REGION Network 4: Diagnostico ASi Global
   // solamente es esta llamada
   RUNG wire#powerrail
      I_Contact( "Activar_Simulador" )
      "FC953_Diagnostico_ASi"(Array_ASI3_C1 := "DB1903_ASI_DIAG".ASI3_GW_C1, Array_ASI3_C2 := "DB1903_ASI_DIAG".ASI3_GW_C2, Array_ASI5_Flags := "DB1903_ASI_DIAG".ASI5_GW_Flags, Error_ASI => "DB1903_ASI_DIAG".ASI_Gateway_Error)
   END_RUNG
   // the same network as SCL:
   IF NOT "Activar_Simulador" THEN
       "FC953_Diagnostico_ASi"(Array_ASI3_C1 := "DB1903_ASI_DIAG".ASI3_GW_C1,
                               Array_ASI3_C2 := "DB1903_ASI_DIAG".ASI3_GW_C2,
                               Array_ASI5_Flags := "DB1903_ASI_DIAG".ASI5_GW_Flags,
                               Error_ASI => "DB1903_ASI_DIAG".ASI_Gateway_Error);
   END_IF;
END_REGION
END_ORGANIZATION_BLOCK

ORGANIZATION_BLOCK "OB82_I/O_FLT1"   // OB82, LAD, DiagnosticErrorInterrupt
TITLE = "I/O Point Fault"
{ S7_Optimized_Access := 'FALSE' }
AUTHOR : ESTANDAR
VERSION : 3.0
// stored: SetENOAutomatically false
   VAR_TEMP
      OB82_EV_CLASS : Byte;   // 16#39, Event class 3, Entering event state, Internal fault event
      OB82_FLT_ID : Byte;   // 16#XX, Fault identifcation code
      OB82_PRIORITY : Byte;   // Priority of OB Execution
      OB82_OB_NUMBR : Byte;   // 82 (Organization block 82, OB82)
      OB82_RESERVED_1 : Byte;   // Reserved for system
      OB82_IO_FLAG : Byte;   // Input (01010100), Output (01010101)
      OB82_MDL_ADDR : Word;   // Base address of module with fault
      OB82_MDL_DEFECT : Bool;   // Module defective
      OB82_INT_FAULT : Bool;   // Internal fault
      OB82_EXT_FAULT : Bool;   // External fault
      OB82_PNT_INFO : Bool;   // Point information
      OB82_EXT_VOLTAGE : Bool;   // External voltage low
      OB82_FLD_CONNCTR : Bool;   // Field wiring connector missing
      OB82_NO_CONFIG : Bool;   // Module has no configuration data
      OB82_CONFIG_ERR : Bool;   // Module has configuration error
      OB82_MDL_TYPE : Byte;   // Type of module
      OB82_SUB_MDL_ERR : Bool;   // Sub-Module is missing or has error
      OB82_COMM_FAULT : Bool;   // Communication fault
      OB82_MDL_STOP : Bool;   // Module is stopped
      OB82_WTCH_DOG_FLT : Bool;   // Watch dog timer stopped module
      OB82_INT_PS_FLT : Bool;   // Internal power supply fault
      OB82_PRIM_BATT_FLT : Bool;   // Primary battery is in fault
      OB82_BCKUP_BATT_FLT : Bool;   // Backup battery is in fault
      OB82_RESERVED_2 : Bool;   // Reserved for system
      OB82_RACK_FLT : Bool;   // Rack fault, only for bus interface module
      OB82_PROC_FLT : Bool;   // Processor fault
      OB82_EPROM_FLT : Bool;   // EPROM fault
      OB82_RAM_FLT : Bool;   // RAM fault
      OB82_ADU_FLT : Bool;   // ADU fault
      OB82_FUSE_FLT : Bool;   // Fuse fault
      OB82_HW_INTR_FLT : Bool;   // Hardware interupt input in fault
      OB82_RESERVED_3 : Bool;   // Reserved for system
      OB82_DATE_TIME : Date_And_Time;   // Date and time OB82 started
   END_VAR
BEGIN
END_ORGANIZATION_BLOCK

ORGANIZATION_BLOCK "OB83_I/O_FLT2"   // OB83, LAD, PullOrPlugOfModules
TITLE = "I/O Point Fault"
{ S7_Optimized_Access := 'FALSE' }
// stored: SetENOAutomatically false
   VAR_TEMP
      OB83_EV_CLASS : Byte;   // 16#38/39, Event class 3, module inserted/removed (8/9)
      OB83_FLT_ID : Byte;   // 16#XX, Fault identifcation code
      OB83_PRIORITY : Byte;   // 26/28 (Priority of 1 is lowest)
      OB83_OB_NUMBR : Byte;   // 83 (Organization block 83, OB83)
      OB83_RESERVED_1 : Byte;   // Reserved for system
      OB83_MDL_ID : Byte;   // Input module (01010100), Output module (01010101)
      OB83_MDL_ADDR : Word;   // Base address of module with point fault
      OB83_RACK_NUM : Word;   // Number of rack that has module with point fault
      OB83_MDL_TYPE : Word;   // Module type with point fault
      OB83_DATE_TIME : Date_And_Time;   // Date and time OB83 started
   END_VAR
BEGIN
END_ORGANIZATION_BLOCK

ORGANIZATION_BLOCK "OB86_ERROR_SLAVES"   // OB86, LAD, RackOrStationFailure
TITLE = "Loss Of Rack Fault"
{ S7_Optimized_Access := 'FALSE' }
AUTHOR : ESTANDAR
VERSION : 3.0
// stored: SetENOAutomatically false
   VAR_TEMP
      OB86_EV_CLASS : Byte;   // 16#38/39 Event class 3
      OB86_FLT_ID : Byte;   // 16#C1/C4/C5, Fault identifcation code
      OB86_PRIORITY : Byte;   // Priority of OB Execution
      OB86_OB_NUMBR : Byte;   // 86 (Organization block 86, OB86)
      OB86_RESERVED_1 : Byte;   // Reserved for system
      OB86_RESERVED_2 : Byte;   // Reserved for system
      OB86_MDL_ADDR : Word;   // Base address of IM module in rack with fault
      OB86_Z23 : DWord;
      OB86_DATE_TIME : Date_And_Time;   // Date and time OB86 started
      P_destino : DWord;
      P_origen : DWord;
      P_infonodo : DWord;
      Numnodo : Word;
      Numred : Word;
      infonodo : Struct
         had_failed : Bool;
         deactivated : Bool;
         reserved_10 : Bool;
         reserved_11 : Bool;
         reserved_12 : Bool;
         reserved_13 : Bool;
         reserved_14 : Bool;
         reserved_15 : Bool;
         OK : Bool;
         maintenance : Bool;
         faulty : Bool;
         failed : Bool;
         was_deactivated : Bool;
         DPV1 : Bool;
         was_under_maintenance : Bool;
         was_failed : Bool;
      END_STRUCT;
   END_VAR
BEGIN
END_ORGANIZATION_BLOCK

FUNCTION_BLOCK "FB420_MesaTL_EtiquetaOrden"   // FB420, LAD
{ S7_Optimized_Access := 'FALSE' }
AUTHOR : ROUTER
NAME : 20180615
VERSION : 3.1
// stored: AutoNumber false, SetENOAutomatically false
   VAR_INPUT
      NumeroMesa : UInt;
      pHsMx : Bool;
      NumSCR : UInt;   // Numero de Scanner asociada a la mesa
      DBFIFO_SCR : UInt;   // DB de Etiquetas Leidas
      LongFIFO_SCR : UInt;   // Numero de Lecturas que se pueden Almacenar
      V_TmpEntrada : Time := T#500MS;
      V_TmpSalida : Time := T#1S;
      MesaDeJDT02 : Bool;
   END_VAR
   VAR_OUTPUT
      PermisoEntrada : Bool;
      PermisoSalida : Bool;
   END_VAR
   VAR
      Mx_ET00 : Bool;
      Mx_ET01 : Bool;
      Mx_ET02 : Bool;
      Mx_ET07 : Bool;
      Mx_ET10 : Bool;
      Mx_ET11 : Bool;
      Mx_ET12 : Bool;
      Mx_ET50 : Bool;
      Mx_ET51 : Bool;
      Mx_ET52 : Bool;
      PresenciaEmiOK : Bool;
      AusenciaEmiOK : Bool;
      BorradoOK : Bool;
      OrdenMx : UInt;
      Motivo : UInt;
      TmpEntrada { S7_SetPoint := 'True'} : TON_TIME;
      TmpSalida { S7_SetPoint := 'True'} : TON_TIME;
      Datos_Scanner { S7_SetPoint := 'True'} : "ROUT_Orden_Fifo_Scanner";
   END_VAR
   VAR_TEMP
      Aux_ET00 : Bool;
      ExisteOrdenSCR : Bool;
      SinOrdenSCR : Bool;
      ExisteOrdenMx : Bool;
      SinOrdenMx : Bool;
      Presencia : Bool;
      Ausencia : Bool;
      Ausencia_especial : Bool;
      MirarOrden : Bool;
      BorradoOrden : Bool;
      Emi_presencia : Bool;
      Emi_ausencia : Bool;
      MesaTMP : UInt;
      MotivoTMP : UInt;
      posicion : Int;
      i : Int;
      longitud : Int;
      codigo_string : String[20];
      mesa_string : String[5];
      moti_string : String[4];
      Mensaje_completo : String;
   END_VAR
BEGIN

REGION Network 1: Incializaciones de la Función
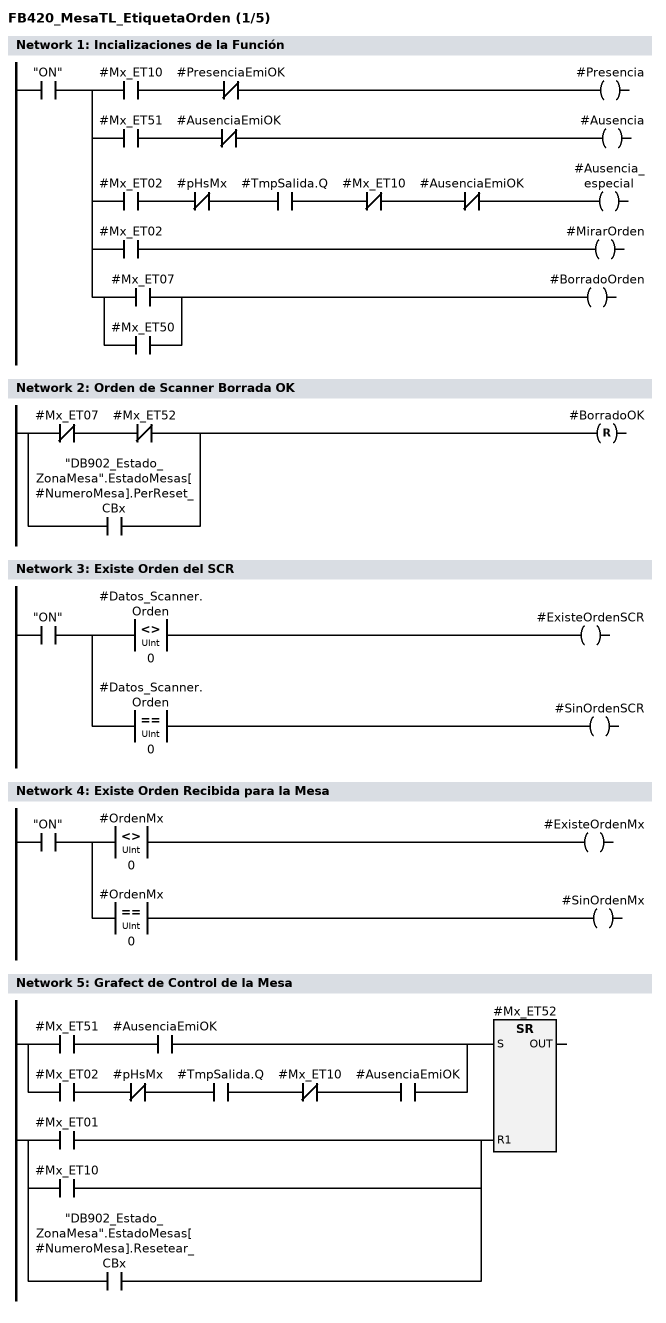
   RUNG wire#powerrail
      Contact( "ON" )
      wire#w1
      Contact( #Mx_ET10 )
      I_Contact( #PresenciaEmiOK )
      Coil( #Presencia )
   END_RUNG
   RUNG wire#w1
      Contact( #Mx_ET51 )
      I_Contact( #AusenciaEmiOK )
      Coil( #Ausencia )
   END_RUNG
   RUNG wire#w1
      Contact( #Mx_ET02 )
      I_Contact( #pHsMx )
      Contact( #TmpSalida.Q )
      I_Contact( #Mx_ET10 )
      I_Contact( #AusenciaEmiOK )
      Coil( #Ausencia_especial )
   END_RUNG
   RUNG wire#w1
      Contact( #Mx_ET02 )
      Coil( #MirarOrden )
   END_RUNG
   RUNG wire#w1
      Contact( #Mx_ET07 )
      wire#w2
      Coil( #BorradoOrden )
   END_RUNG
   RUNG wire#w1
      Contact( #Mx_ET50 )
   END_RUNG wire#w2
   // the same network as SCL:
   #Presencia := "ON" AND #Mx_ET10 AND NOT #PresenciaEmiOK;
   #Ausencia := "ON" AND #Mx_ET51 AND NOT #AusenciaEmiOK;
   #Ausencia_especial := "ON" AND #Mx_ET02 AND NOT #pHsMx AND #TmpSalida.Q AND NOT #Mx_ET10 AND NOT #AusenciaEmiOK;
   #MirarOrden := "ON" AND #Mx_ET02;
   #BorradoOrden := "ON" AND (#Mx_ET07 OR #Mx_ET50);
END_REGION

REGION Network 2: Orden de Scanner Borrada OK
   RUNG wire#powerrail
      I_Contact( #Mx_ET07 )
      I_Contact( #Mx_ET52 )
      wire#w1
      R_Coil( #BorradoOK )
   END_RUNG
   RUNG wire#powerrail
      Contact( "DB902_Estado_ZonaMesa".EstadoMesas[#NumeroMesa].PerReset_CBx )
   END_RUNG wire#w1
   // the same network as SCL:
   IF (NOT #Mx_ET07 AND NOT #Mx_ET52) OR "DB902_Estado_ZonaMesa".EstadoMesas[#NumeroMesa].PerReset_CBx THEN
       #BorradoOK := FALSE;
   END_IF;
END_REGION

REGION Network 3: Existe Orden del SCR
   RUNG wire#powerrail
      Contact( "ON" )
      wire#w1
      { S7_Templates := "SrcType := UInt" } NE_Contact(in1 := #Datos_Scanner.Orden, in2 := 0)
      Coil( #ExisteOrdenSCR )
   END_RUNG
   RUNG wire#w1
      { S7_Templates := "SrcType := UInt" } EQ_Contact(in1 := #Datos_Scanner.Orden, in2 := 0)
      Coil( #SinOrdenSCR )
   END_RUNG
   // the same network as SCL:
   #ExisteOrdenSCR := "ON" AND (#Datos_Scanner.Orden <> 0);
   #SinOrdenSCR := "ON" AND (#Datos_Scanner.Orden = 0);
END_REGION

REGION Network 4: Existe Orden Recibida para la Mesa
   RUNG wire#powerrail
      Contact( "ON" )
      wire#w1
      { S7_Templates := "SrcType := UInt" } NE_Contact(in1 := #OrdenMx, in2 := 0)
      Coil( #ExisteOrdenMx )
   END_RUNG
   RUNG wire#w1
      { S7_Templates := "SrcType := UInt" } EQ_Contact(in1 := #OrdenMx, in2 := 0)
      Coil( #SinOrdenMx )
   END_RUNG
   // the same network as SCL:
   #ExisteOrdenMx := "ON" AND (#OrdenMx <> 0);
   #SinOrdenMx := "ON" AND (#OrdenMx = 0);
END_REGION

REGION Network 5: Grafect de Control de la Mesa
   RUNG wire#powerrail
      Contact( #Mx_ET51 )
      Contact( #AusenciaEmiOK )
      wire#w1
      S_SR(operand := #Mx_ET52, r1 := wire#w2)
   END_RUNG
   RUNG wire#powerrail
      Contact( #Mx_ET02 )
      I_Contact( #pHsMx )
      Contact( #TmpSalida.Q )
      I_Contact( #Mx_ET10 )
      Contact( #AusenciaEmiOK )
   END_RUNG wire#w1
   RUNG wire#powerrail
      Contact( #Mx_ET01 )
   END_RUNG wire#w2
   RUNG wire#powerrail
      Contact( #Mx_ET10 )
   END_RUNG wire#w2
   RUNG wire#powerrail
      Contact( "DB902_Estado_ZonaMesa".EstadoMesas[#NumeroMesa].Resetear_CBx )
   END_RUNG wire#w2
   // the same network as SCL:
   IF (#Mx_ET51 AND #AusenciaEmiOK) OR (#Mx_ET02 AND NOT #pHsMx AND #TmpSalida.Q AND NOT #Mx_ET10 AND #AusenciaEmiOK) THEN
       #Mx_ET52 := TRUE;   // SR flip-flop
   END_IF;
   IF #Mx_ET01 OR #Mx_ET10 OR "DB902_Estado_ZonaMesa".EstadoMesas[#NumeroMesa].Resetear_CBx THEN
       #Mx_ET52 := FALSE;
   END_IF;
END_REGION

REGION Network 6
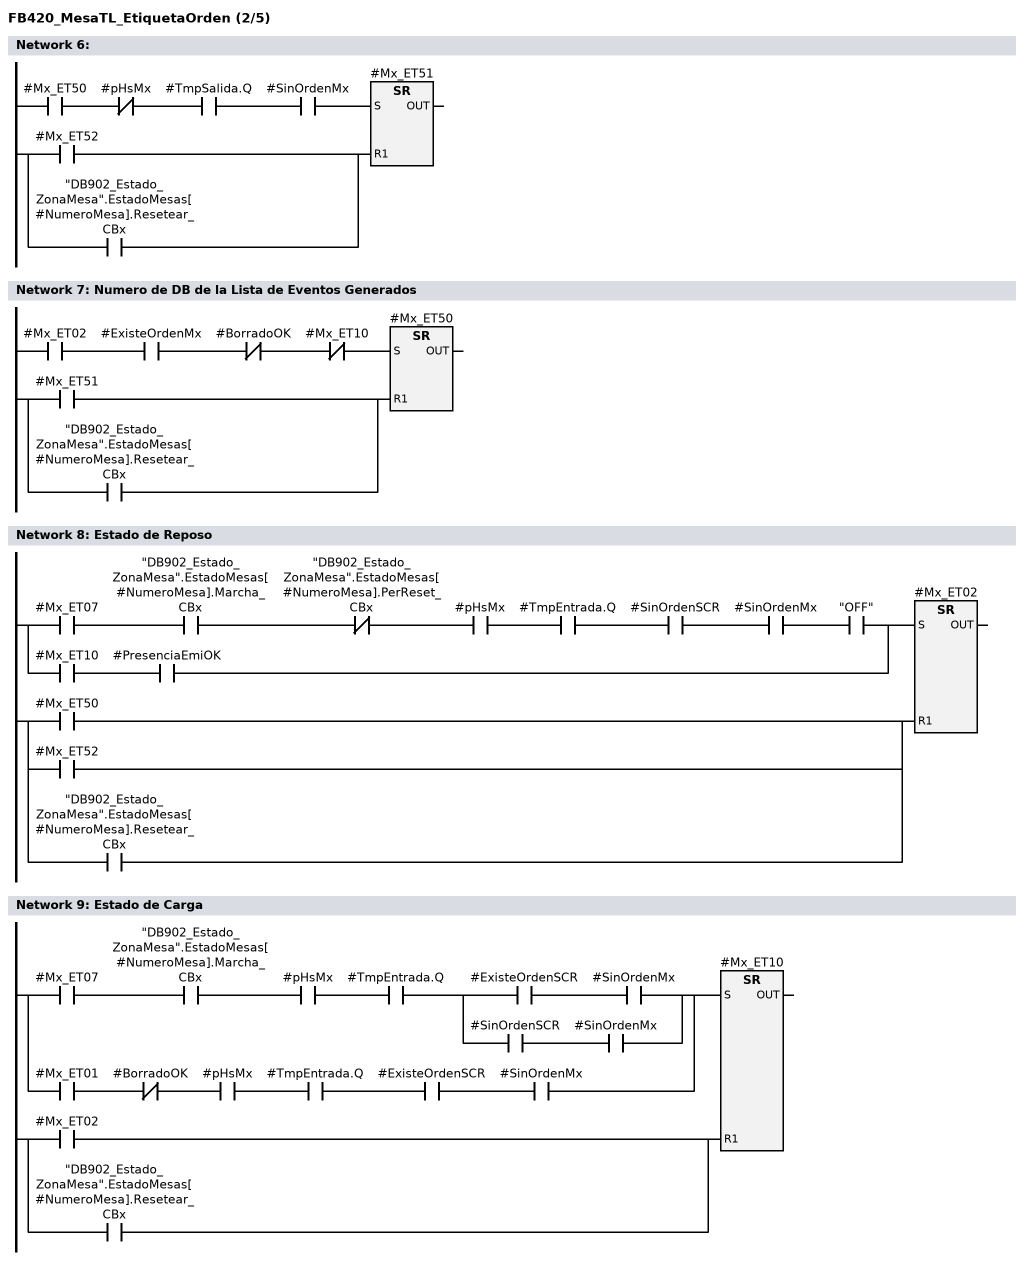
   RUNG wire#powerrail
      Contact( #Mx_ET50 )
      I_Contact( #pHsMx )
      Contact( #TmpSalida.Q )
      Contact( #SinOrdenMx )
      S_SR(operand := #Mx_ET51, r1 := wire#w1)
   END_RUNG
   RUNG wire#powerrail
      Contact( #Mx_ET52 )
   END_RUNG wire#w1
   RUNG wire#powerrail
      Contact( "DB902_Estado_ZonaMesa".EstadoMesas[#NumeroMesa].Resetear_CBx )
   END_RUNG wire#w1
   // the same network as SCL:
   IF #Mx_ET50 AND NOT #pHsMx AND #TmpSalida.Q AND #SinOrdenMx THEN
       #Mx_ET51 := TRUE;   // SR flip-flop
   END_IF;
   IF #Mx_ET52 OR "DB902_Estado_ZonaMesa".EstadoMesas[#NumeroMesa].Resetear_CBx THEN
       #Mx_ET51 := FALSE;
   END_IF;
END_REGION

REGION Network 7: Numero de DB de la Lista de Eventos Generados
   RUNG wire#powerrail
      Contact( #Mx_ET02 )
      Contact( #ExisteOrdenMx )
      I_Contact( #BorradoOK )
      I_Contact( #Mx_ET10 )
      S_SR(operand := #Mx_ET50, r1 := wire#w1)
   END_RUNG
   RUNG wire#powerrail
      Contact( #Mx_ET51 )
   END_RUNG wire#w1
   RUNG wire#powerrail
      Contact( "DB902_Estado_ZonaMesa".EstadoMesas[#NumeroMesa].Resetear_CBx )
   END_RUNG wire#w1
   // the same network as SCL:
   IF #Mx_ET02 AND #ExisteOrdenMx AND NOT #BorradoOK AND NOT #Mx_ET10 THEN
       #Mx_ET50 := TRUE;   // SR flip-flop
   END_IF;
   IF #Mx_ET51 OR "DB902_Estado_ZonaMesa".EstadoMesas[#NumeroMesa].Resetear_CBx THEN
       #Mx_ET50 := FALSE;
   END_IF;
END_REGION

REGION Network 8: Estado de Reposo
   RUNG wire#powerrail
      Contact( #Mx_ET07 )
      Contact( "DB902_Estado_ZonaMesa".EstadoMesas[#NumeroMesa].Marcha_CBx )
      I_Contact( "DB902_Estado_ZonaMesa".EstadoMesas[#NumeroMesa].PerReset_CBx )
      Contact( #pHsMx )
      Contact( #TmpEntrada.Q )
      Contact( #SinOrdenSCR )
      Contact( #SinOrdenMx )
      Contact( "OFF" )
      wire#w1
      S_SR(operand := #Mx_ET02, r1 := wire#w2)
   END_RUNG
   RUNG wire#powerrail
      Contact( #Mx_ET10 )
      Contact( #PresenciaEmiOK )
   END_RUNG wire#w1
   RUNG wire#powerrail
      Contact( #Mx_ET50 )
   END_RUNG wire#w2
   RUNG wire#powerrail
      Contact( #Mx_ET52 )
   END_RUNG wire#w2
   RUNG wire#powerrail
      Contact( "DB902_Estado_ZonaMesa".EstadoMesas[#NumeroMesa].Resetear_CBx )
   END_RUNG wire#w2
   // the same network as SCL:
   IF (#Mx_ET07 AND "DB902_Estado_ZonaMesa".EstadoMesas[#NumeroMesa].Marcha_CBx AND NOT "DB902_Estado_ZonaMesa".EstadoMesas[#NumeroMesa].PerReset_CBx AND #pHsMx AND #TmpEntrada.Q AND #SinOrdenSCR AND #SinOrdenMx AND "OFF") OR (#Mx_ET10 AND #PresenciaEmiOK) THEN
       #Mx_ET02 := TRUE;   // SR flip-flop
   END_IF;
   IF #Mx_ET50 OR #Mx_ET52 OR "DB902_Estado_ZonaMesa".EstadoMesas[#NumeroMesa].Resetear_CBx THEN
       #Mx_ET02 := FALSE;
   END_IF;
END_REGION

REGION Network 9: Estado de Carga
   RUNG wire#powerrail
      Contact( #Mx_ET07 )
      Contact( "DB902_Estado_ZonaMesa".EstadoMesas[#NumeroMesa].Marcha_CBx )
      Contact( #pHsMx )
      Contact( #TmpEntrada.Q )
      wire#w1
      Contact( #ExisteOrdenSCR )
      Contact( #SinOrdenMx )
      wire#w2
      S_SR(operand := #Mx_ET10, r1 := wire#w3)
   END_RUNG
   RUNG wire#w1
      Contact( #SinOrdenSCR )
      Contact( #SinOrdenMx )
   END_RUNG wire#w2
   RUNG wire#powerrail
      Contact( #Mx_ET01 )
      I_Contact( #BorradoOK )
      Contact( #pHsMx )
      Contact( #TmpEntrada.Q )
      Contact( #ExisteOrdenSCR )
      Contact( #SinOrdenMx )
   END_RUNG wire#w2
   RUNG wire#powerrail
      Contact( #Mx_ET02 )
   END_RUNG wire#w3
   RUNG wire#powerrail
      Contact( "DB902_Estado_ZonaMesa".EstadoMesas[#NumeroMesa].Resetear_CBx )
   END_RUNG wire#w3
   // the same network as SCL:
   IF (#Mx_ET07 AND "DB902_Estado_ZonaMesa".EstadoMesas[#NumeroMesa].Marcha_CBx AND #pHsMx AND #TmpEntrada.Q AND ((#ExisteOrdenSCR AND #SinOrdenMx) OR (#SinOrdenSCR AND #SinOrdenMx))) OR (#Mx_ET01 AND NOT #BorradoOK AND #pHsMx AND #TmpEntrada.Q AND #ExisteOrdenSCR AND #SinOrdenMx) THEN
       #Mx_ET10 := TRUE;   // SR flip-flop
   END_IF;
   IF #Mx_ET02 OR "DB902_Estado_ZonaMesa".EstadoMesas[#NumeroMesa].Resetear_CBx THEN
       #Mx_ET10 := FALSE;
   END_IF;
END_REGION

REGION Network 10: Estado de Vacia
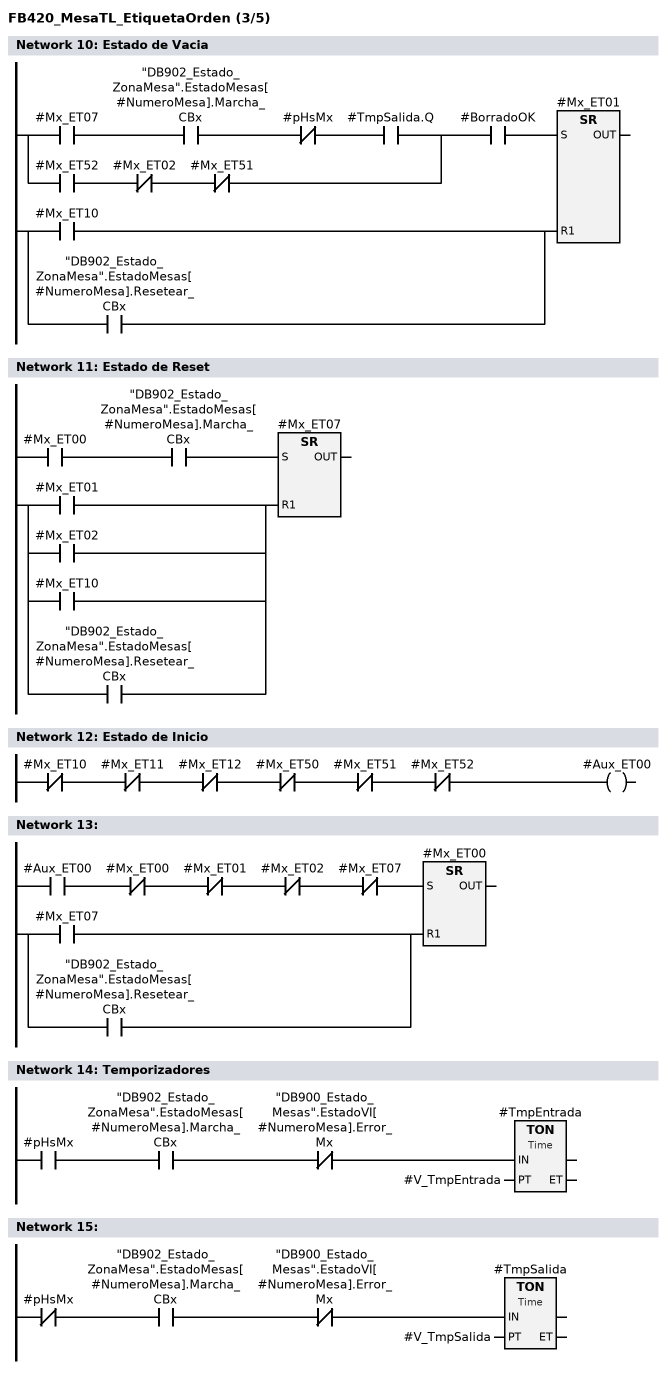
   RUNG wire#powerrail
      Contact( #Mx_ET07 )
      Contact( "DB902_Estado_ZonaMesa".EstadoMesas[#NumeroMesa].Marcha_CBx )
      I_Contact( #pHsMx )
      Contact( #TmpSalida.Q )
      wire#w1
      Contact( #BorradoOK )
      S_SR(operand := #Mx_ET01, r1 := wire#w2)
   END_RUNG
   RUNG wire#powerrail
      Contact( #Mx_ET52 )
      I_Contact( #Mx_ET02 )
      I_Contact( #Mx_ET51 )
   END_RUNG wire#w1
   RUNG wire#powerrail
      Contact( #Mx_ET10 )
   END_RUNG wire#w2
   RUNG wire#powerrail
      Contact( "DB902_Estado_ZonaMesa".EstadoMesas[#NumeroMesa].Resetear_CBx )
   END_RUNG wire#w2
   // the same network as SCL:
   IF ((#Mx_ET07 AND "DB902_Estado_ZonaMesa".EstadoMesas[#NumeroMesa].Marcha_CBx AND NOT #pHsMx AND #TmpSalida.Q) OR (#Mx_ET52 AND NOT #Mx_ET02 AND NOT #Mx_ET51)) AND #BorradoOK THEN
       #Mx_ET01 := TRUE;   // SR flip-flop
   END_IF;
   IF #Mx_ET10 OR "DB902_Estado_ZonaMesa".EstadoMesas[#NumeroMesa].Resetear_CBx THEN
       #Mx_ET01 := FALSE;
   END_IF;
END_REGION

REGION Network 11: Estado de Reset
   RUNG wire#powerrail
      Contact( #Mx_ET00 )
      Contact( "DB902_Estado_ZonaMesa".EstadoMesas[#NumeroMesa].Marcha_CBx )
      S_SR(operand := #Mx_ET07, r1 := wire#w1)
   END_RUNG
   RUNG wire#powerrail
      Contact( #Mx_ET01 )
   END_RUNG wire#w1
   RUNG wire#powerrail
      Contact( #Mx_ET02 )
   END_RUNG wire#w1
   RUNG wire#powerrail
      Contact( #Mx_ET10 )
   END_RUNG wire#w1
   RUNG wire#powerrail
      Contact( "DB902_Estado_ZonaMesa".EstadoMesas[#NumeroMesa].Resetear_CBx )
   END_RUNG wire#w1
   // the same network as SCL:
   IF #Mx_ET00 AND "DB902_Estado_ZonaMesa".EstadoMesas[#NumeroMesa].Marcha_CBx THEN
       #Mx_ET07 := TRUE;   // SR flip-flop
   END_IF;
   IF #Mx_ET01 OR #Mx_ET02 OR #Mx_ET10 OR "DB902_Estado_ZonaMesa".EstadoMesas[#NumeroMesa].Resetear_CBx THEN
       #Mx_ET07 := FALSE;
   END_IF;
END_REGION

REGION Network 12: Estado de Inicio
   RUNG wire#powerrail
      I_Contact( #Mx_ET10 )
      I_Contact( #Mx_ET11 )
      I_Contact( #Mx_ET12 )
      I_Contact( #Mx_ET50 )
      I_Contact( #Mx_ET51 )
      I_Contact( #Mx_ET52 )
      Coil( #Aux_ET00 )
   END_RUNG
   // the same network as SCL:
   #Aux_ET00 := NOT #Mx_ET10 AND NOT #Mx_ET11 AND NOT #Mx_ET12 AND NOT #Mx_ET50 AND NOT #Mx_ET51 AND NOT #Mx_ET52;
END_REGION

REGION Network 13
   RUNG wire#powerrail
      Contact( #Aux_ET00 )
      I_Contact( #Mx_ET00 )
      I_Contact( #Mx_ET01 )
      I_Contact( #Mx_ET02 )
      I_Contact( #Mx_ET07 )
      S_SR(operand := #Mx_ET00, r1 := wire#w1)
   END_RUNG
   RUNG wire#powerrail
      Contact( #Mx_ET07 )
   END_RUNG wire#w1
   RUNG wire#powerrail
      Contact( "DB902_Estado_ZonaMesa".EstadoMesas[#NumeroMesa].Resetear_CBx )
   END_RUNG wire#w1
   // the same network as SCL:
   IF #Aux_ET00 AND NOT #Mx_ET00 AND NOT #Mx_ET01 AND NOT #Mx_ET02 AND NOT #Mx_ET07 THEN
       #Mx_ET00 := TRUE;   // SR flip-flop
   END_IF;
   IF #Mx_ET07 OR "DB902_Estado_ZonaMesa".EstadoMesas[#NumeroMesa].Resetear_CBx THEN
       #Mx_ET00 := FALSE;
   END_IF;
END_REGION

REGION Network 14: Temporizadores
   RUNG wire#powerrail
      Contact( #pHsMx )
      Contact( "DB902_Estado_ZonaMesa".EstadoMesas[#NumeroMesa].Marcha_CBx )
      I_Contact( "DB900_Estado_Mesas".EstadoVI[#NumeroMesa].Error_Mx )
      { S7_Templates := "time_type := Time" } #TmpEntrada.TON(pt := #V_TmpEntrada, et =>)
   END_RUNG
   // the same network as SCL:
   #TmpEntrada(IN := #pHsMx AND "DB902_Estado_ZonaMesa".EstadoMesas[#NumeroMesa].Marcha_CBx AND NOT "DB900_Estado_Mesas".EstadoVI[#NumeroMesa].Error_Mx,   // TON
               PT := #V_TmpEntrada);
END_REGION

REGION Network 15
   RUNG wire#powerrail
      I_Contact( #pHsMx )
      Contact( "DB902_Estado_ZonaMesa".EstadoMesas[#NumeroMesa].Marcha_CBx )
      I_Contact( "DB900_Estado_Mesas".EstadoVI[#NumeroMesa].Error_Mx )
      { S7_Templates := "time_type := Time" } #TmpSalida.TON(pt := #V_TmpSalida, et =>)
   END_RUNG
   // the same network as SCL:
   #TmpSalida(IN := NOT #pHsMx AND "DB902_Estado_ZonaMesa".EstadoMesas[#NumeroMesa].Marcha_CBx AND NOT "DB900_Estado_Mesas".EstadoVI[#NumeroMesa].Error_Mx,   // TON
              PT := #V_TmpSalida);
END_REGION

REGION Network 16: Eliminar la Lectura de Scanner
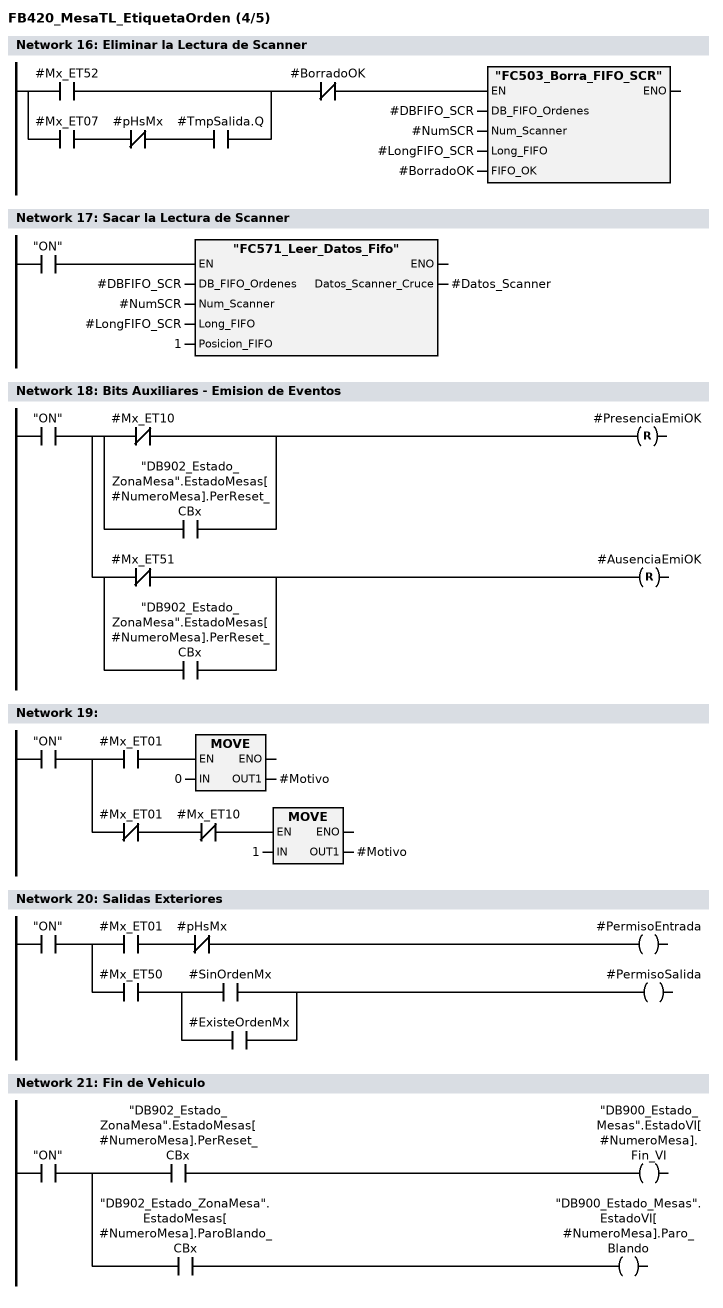
   RUNG wire#powerrail
      Contact( #Mx_ET52 )
      wire#w1
      I_Contact( #BorradoOK )
      "FC503_Borra_FIFO_SCR"(DB_FIFO_Ordenes := #DBFIFO_SCR, Num_Scanner := #NumSCR, Long_FIFO := #LongFIFO_SCR, FIFO_OK := #BorradoOK)
   END_RUNG
   RUNG wire#powerrail
      Contact( #Mx_ET07 )
      I_Contact( #pHsMx )
      Contact( #TmpSalida.Q )
   END_RUNG wire#w1
   // the same network as SCL:
   IF (#Mx_ET52 OR (#Mx_ET07 AND NOT #pHsMx AND #TmpSalida.Q)) AND NOT #BorradoOK THEN
       "FC503_Borra_FIFO_SCR"(DB_FIFO_Ordenes := #DBFIFO_SCR,
                              Num_Scanner := #NumSCR,
                              Long_FIFO := #LongFIFO_SCR,
                              FIFO_OK := #BorradoOK);
   END_IF;
END_REGION

REGION Network 17: Sacar la Lectura de Scanner
   RUNG wire#powerrail
      Contact( "ON" )
      "FC571_Leer_Datos_Fifo"(DB_FIFO_Ordenes := #DBFIFO_SCR, Num_Scanner := #NumSCR, Long_FIFO := #LongFIFO_SCR, Posicion_FIFO := 1, Datos_Scanner_Cruce => #Datos_Scanner)
   END_RUNG
   // the same network as SCL:
   IF "ON" THEN
       "FC571_Leer_Datos_Fifo"(DB_FIFO_Ordenes := #DBFIFO_SCR,
                               Num_Scanner := #NumSCR,
                               Long_FIFO := #LongFIFO_SCR,
                               Posicion_FIFO := 1,
                               Datos_Scanner_Cruce => #Datos_Scanner);
   END_IF;
END_REGION

REGION Network 18: Bits Auxiliares - Emision de Eventos
   RUNG wire#powerrail
      Contact( "ON" )
      wire#w1
      I_Contact( #Mx_ET10 )
      wire#w2
      R_Coil( #PresenciaEmiOK )
   END_RUNG
   RUNG wire#w1
      Contact( "DB902_Estado_ZonaMesa".EstadoMesas[#NumeroMesa].PerReset_CBx )
   END_RUNG wire#w2
   RUNG wire#w1
      I_Contact( #Mx_ET51 )
      wire#w3
      R_Coil( #AusenciaEmiOK )
   END_RUNG
   RUNG wire#w1
      Contact( "DB902_Estado_ZonaMesa".EstadoMesas[#NumeroMesa].PerReset_CBx )
   END_RUNG wire#w3
   // the same network as SCL:
   IF "ON" AND (NOT #Mx_ET10 OR "DB902_Estado_ZonaMesa".EstadoMesas[#NumeroMesa].PerReset_CBx) THEN
       #PresenciaEmiOK := FALSE;
   END_IF;
   IF "ON" AND (NOT #Mx_ET51 OR "DB902_Estado_ZonaMesa".EstadoMesas[#NumeroMesa].PerReset_CBx) THEN
       #AusenciaEmiOK := FALSE;
   END_IF;
END_REGION

REGION Network 19
   RUNG wire#powerrail
      Contact( "ON" )
      wire#w1
      Contact( #Mx_ET01 )
      { S7_GenerateENO := "TRUE" } Move(in := 0, out1 => #Motivo)
   END_RUNG
   RUNG wire#w1
      I_Contact( #Mx_ET01 )
      I_Contact( #Mx_ET10 )
      { S7_GenerateENO := "TRUE" } Move(in := 1, out1 => #Motivo)
   END_RUNG
   // the same network as SCL:
   IF "ON" AND #Mx_ET01 THEN #Motivo := 0; END_IF;
   IF "ON" AND NOT #Mx_ET01 AND NOT #Mx_ET10 THEN #Motivo := 1; END_IF;
END_REGION

REGION Network 20: Salidas Exteriores
   RUNG wire#powerrail
      Contact( "ON" )
      wire#w1
      Contact( #Mx_ET01 )
      I_Contact( #pHsMx )
      Coil( #PermisoEntrada )
   END_RUNG
   RUNG wire#w1
      Contact( #Mx_ET50 )
      wire#w2
      Contact( #SinOrdenMx )
      wire#w3
      Coil( #PermisoSalida )
   END_RUNG
   RUNG wire#w2
      Contact( #ExisteOrdenMx )
   END_RUNG wire#w3
   // the same network as SCL:
   #PermisoEntrada := "ON" AND #Mx_ET01 AND NOT #pHsMx;
   #PermisoSalida := "ON" AND #Mx_ET50 AND (#SinOrdenMx OR #ExisteOrdenMx);
END_REGION

REGION Network 21: Fin de Vehiculo
   RUNG wire#powerrail
      Contact( "ON" )
      wire#w1
      Contact( "DB902_Estado_ZonaMesa".EstadoMesas[#NumeroMesa].PerReset_CBx )
      Coil( "DB900_Estado_Mesas".EstadoVI[#NumeroMesa].Fin_VI )
   END_RUNG
   RUNG wire#w1
      Contact( "DB902_Estado_ZonaMesa".EstadoMesas[#NumeroMesa].ParoBlando_CBx )
      Coil( "DB900_Estado_Mesas".EstadoVI[#NumeroMesa].Paro_Blando )
   END_RUNG
   // the same network as SCL:
   "DB900_Estado_Mesas".EstadoVI[#NumeroMesa].Fin_VI := "ON" AND "DB902_Estado_ZonaMesa".EstadoMesas[#NumeroMesa].PerReset_CBx;
   "DB900_Estado_Mesas".EstadoVI[#NumeroMesa].Paro_Blando := "ON" AND "DB902_Estado_ZonaMesa".EstadoMesas[#NumeroMesa].ParoBlando_CBx;
END_REGION

REGION Network 22
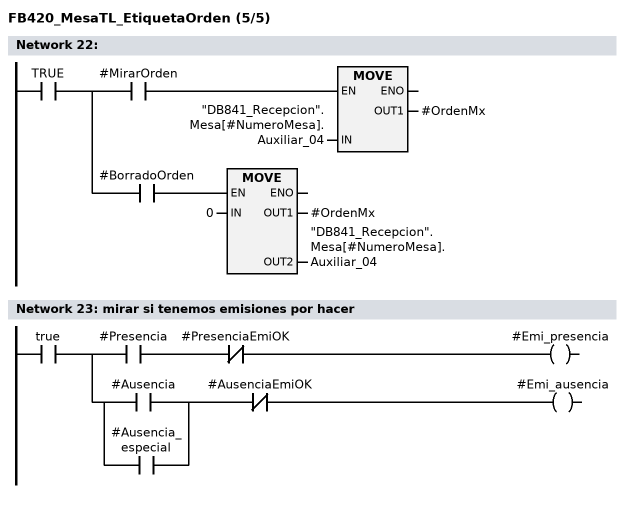
   RUNG wire#powerrail
      Contact( TRUE )
      wire#w1
      Contact( #MirarOrden )
      Move(in := "DB841_Recepcion".Mesa[#NumeroMesa].Auxiliar_04, out1 => #OrdenMx)
   END_RUNG
   RUNG wire#w1
      Contact( #BorradoOrden )
      Move(in := 0, out1 => #OrdenMx, out2 => "DB841_Recepcion".Mesa[#NumeroMesa].Auxiliar_04)
   END_RUNG
   // the same network as SCL:
   IF TRUE AND #MirarOrden THEN #OrdenMx := "DB841_Recepcion".Mesa[#NumeroMesa].Auxiliar_04; END_IF;
   IF TRUE AND #BorradoOrden THEN
       #OrdenMx := 0;
       "DB841_Recepcion".Mesa[#NumeroMesa].Auxiliar_04 := 0;
   END_IF;
END_REGION

REGION Network 23: mirar si tenemos emisiones por hacer
   RUNG wire#powerrail
      Contact( true )
      wire#w1
      Contact( #Presencia )
      I_Contact( #PresenciaEmiOK )
      Coil( #Emi_presencia )
   END_RUNG
   RUNG wire#w1
      Contact( #Ausencia )
      wire#w2
      I_Contact( #AusenciaEmiOK )
      Coil( #Emi_ausencia )
   END_RUNG
   RUNG wire#w1
      Contact( #Ausencia_especial )
   END_RUNG wire#w2
   // the same network as SCL:
   #Emi_presencia := true AND #Presencia AND NOT #PresenciaEmiOK;
   #Emi_ausencia := true AND (#Ausencia OR #Ausencia_especial) AND NOT #AusenciaEmiOK;
END_REGION

REGION Network 24 (SCL)
   IF (#Emi_presencia = true) OR (#Emi_ausencia = true) THEN
       #MesaTMP := #NumeroMesa + "CTE_OffsetMesa";
       #MotivoTMP := #Motivo;
   ELSE
       RETURN;
   END_IF;
END_REGION

REGION Network 25 (SCL)
   //miramos si tenemos que emitir el evento al JDT1 o al JDT2 para buscar hueco
   IF #MesaDeJDT02 = true THEN
   REGION buscar en JDT2

       #posicion := -1;
       FOR #i := 0 TO 100 BY 1 DO
           #longitud := LEN("DB197_eventos_generados_routing_JDT2".evento[#i]);
           IF #longitud = 0 THEN
               #posicion := #i;
               EXIT;
           END_IF;
       END_FOR;

       // si no hay sitio para escribir salimos del bloque
       IF #posicion = -1 THEN
           RETURN;
       END_IF;
   END_REGION
   ;
   ELSE
       REGION buscar en JDT1

           #posicion := -1;
           FOR #i := 0 TO 100 BY 1 DO
               #longitud := LEN("DB198_eventos_generados_routing_JDT1".evento[#i]);
               IF #longitud = 0 THEN
                   #posicion := #i;
                   EXIT;
               END_IF;
           END_FOR;

           // si no hay sitio para escribir salimos del bloque
           IF #posicion = -1 THEN
               RETURN;
           END_IF;
       END_REGION
   END_IF;


   // si continuamos es porque podemos formatear el mensaje
   // 




   #mesa_string := DELETE(IN := (UINT_TO_STRING(IN := #MesaTMP )), L := 1, P := 1);
   #codigo_string := DELETE(IN := (ULINT_TO_STRING(IN := #Datos_Scanner.Identificador)), L := 1, P := 1);

   // CODIFICACION DEL MOTIVO
   #moti_string := '----'; // INICIALIAMOS A ESTE VALOR POR SI ACASO

   IF ((#Emi_presencia=TRUE)AND(#MotivoTMP= 0)) THEN
       #moti_string := 'NORM';
   ELSIF((#Emi_presencia=TRUE)AND(#MotivoTMP= 1)) THEN
       #moti_string := 'RESE';
   ELSIF((#Emi_ausencia=TRUE)AND(#Ausencia_especial=FALSE)) THEN
       #moti_string := 'NORM';
   ELSIF((#Emi_ausencia=TRUE)AND(#Ausencia_especial=TRUE)) THEN
       #moti_string := 'FAIL';
   END_IF;



   // aqui formateamos el mensaje que toca presencia, ausencia o ausencia especial

   IF #Emi_presencia = true THEN
       #Mensaje_completo:= CONCAT(IN1 := '{PRES[MESA]', IN2 := #mesa_string, IN3 := '[SSCC]', IN4 := #codigo_string, IN5 := '[MOTI]', IN6 := #moti_string,IN7:="DB921_DATOS_FECHA_HORA".TIME_STAMP,IN8:='}');
       #PresenciaEmiOK := TRUE;
   ELSIF #Emi_ausencia = TRUE THEN
       #Mensaje_completo := CONCAT(IN1 := '{AUSE[MESA]', IN2 := #mesa_string, IN3 := '[SSCC]', IN4 := #codigo_string, IN5 := '[MOTI]', IN6 := #moti_string,IN7:="DB921_DATOS_FECHA_HORA".TIME_STAMP,IN8:='}');
       #AusenciaEmiOK := TRUE;
   END_IF;

   // ESCRIBIMOS EN EL DB DE EMISIÓN DEL jdt QUE CORRESPONDE
   // 
   IF #MesaDeJDT02 = true THEN

       "DB197_eventos_generados_routing_JDT2".evento[#posicion] := #Mensaje_completo;
   ELSE
       "DB198_eventos_generados_routing_JDT1".evento[#posicion] := #Mensaje_completo;

   END_IF;
END_REGION
END_FUNCTION_BLOCK

FUNCTION "FC571_Leer_Datos_Fifo" : Void   // FC571, STL
{ S7_Optimized_Access := 'FALSE' }
// stored: AutoNumber false
   VAR_INPUT
      DB_FIFO_Ordenes : UInt;
      Num_Scanner : UInt;   // Numero de scanner sobre el que se realiza la busqueda
      Long_FIFO : UInt;
      Posicion_FIFO : UInt;
   END_VAR
   VAR_OUTPUT
      Datos_Scanner_Cruce : "ROUT_Orden_Fifo_Scanner";
   END_VAR
   VAR_TEMP
      Guardar_AR2 : DWord;
      P_Inicio_Datos : DWord;
      P_Any_Datos : Any;
      NumDB : Word;
      MaxRegistros : UInt;
      LongRegistro : UInt;
      OffsetPrimerRegistro : UInt;
      ValorReturn : Int;
      Elementos_X_Registro : Int;
      Relleno : Byte;
   END_VAR
BEGIN

NETWORK
TITLE = Inicializar Variables
//////////////////////////////////////////////////////////////////////////
/// - Datos del DB a leer

      L     #DB_FIFO_Ordenes;  // - Numero de DB a Leer
      T     #NumDB;
      L     "CTE_MaxMesas";  // - Numero Maximo de Registros
      T     #MaxRegistros;
      L     "ROUT_Long_Reg_Datos_FIFO";  // - Longitud de la estructura del Registro
      T     #LongRegistro;
      L     #Long_FIFO;
      T     #Elementos_X_Registro;
      L     0;  // - Offset del Primer Registro
      T     #OffsetPrimerRegistro;


//////////////////////////////////////////////////////////////////////////
/// - Inicilizar Registro de Salida

      L     0;
      T     #Relleno;

      CALL  FILL
      ( BVAL    := #Relleno,
        RET_VAL := #ValorReturn,
        BLK     := #Datos_Scanner_Cruce
      );



NETWORK
TITLE = Posicionarse en el Registro
//////////////////////////////////////////////////////////////////////////
/// - Comprobar si el registro existe (Maximo de Registros)

      L     #Num_Scanner;
      L     #MaxRegistros;
      >I;
      JC    Error_MaxRegistros;


//////////////////////////////////////////////////////////////////////////
/// - Calculo de la posicion del registro

// primero nos posicionamos en el primer elemento de la fifo

      L     #Num_Scanner;
      L     #LongRegistro;
      *I;
      L     #Elementos_X_Registro;
      *I;
      L     #OffsetPrimerRegistro;
      +I;
      SLD   3;
      T     #P_Inicio_Datos;

// miramos si tenemos que sacar un registro diferente del primero

      L     #Posicion_FIFO;
      L     1;
      ==I;
      JC    sacar_datos;
// si es un registro diferente del primero, calculamos el offset para colocarnos en el registro correcto

      L     #Posicion_FIFO;
      L     1;
      -I;
      L     #LongRegistro;
      *I;
      SLD   3;
      L     #P_Inicio_Datos;
      +D;
      T     #P_Inicio_Datos;


NETWORK
TITLE = Transferenica del Registro
//////////////////////////////////////////////////////////////////////////
/// - Calculo del Puntero Any de los Datos
sacar_datos:NOP   0;
      TAR2  #Guardar_AR2;  // - Guardar el Puntero AR2

      LAR2  P##P_Any_Datos;  // - Direccion del Puntero Any
      L     B#16#10;  //   10H para S7
      T     LB [AR2, P#0.0];
      L     B#16#2;  //   Tipo de Datos (BYTE)
      T     LB [AR2, P#1.0];
      L     #LongRegistro;  //   Longitud de la Estructura
      T     LW [AR2, P#2.0];
      L     #NumDB;  //   Numero de DB
      T     LW [AR2, P#4.0];
      L     #P_Inicio_Datos;  //   Direccion de Inicio
      T     LD [AR2, P#6.0];
      L     B#16#84;  //   El Area de Memoria = DB
      T     LB [AR2, P#6.0];

      LAR2  #Guardar_AR2;  // - Recuperar el Puntero AR2

//////////////////////////////////////////////////////////////////////////
/// - Transferencia de los Datos a Leer

      CALL  BLKMOV
      ( SRCBLK  := #P_Any_Datos,
        RET_VAL := #ValorReturn,
        DSTBLK  := #Datos_Scanner_Cruce
      );

      L     #ValorReturn;  // - Comprobar que se ha leido el registro
      L     0;
      <>I;
      JC    Error_LecturaDelRegisto;


//////////////////////////////////////////////////////////////////////////
/// - Fin de la Lectura del Registro

      BE;  // - Finalizar bloque



NETWORK
TITLE = Errores en el Sistema de Lectura
//////////////////////////////////////////////////////////////////////////
/// - Numero De Maximo de Registros Sobrepasado

Error_MaxRegistros:NOP   0;
      BE;  // - Finalizar bloque

////////////////////////////////////////////////////
/// - Error a Leer el Registro

Error_LecturaDelRegisto:NOP   0;
      BE;  // - Finalizar bloque


END_FUNCTION

FUNCTION "FC499_Mirar_Estado_Vacio" : Void   // FC499, LAD
{ S7_Optimized_Access := 'FALSE' }
AUTHOR : TLigero
NAME : 20150226
VERSION : 3.0
// stored: AutoNumber false, SetENOAutomatically false
   VAR_INPUT
      Numero_Mesa_Ini : UInt;
      Numero_Mesa_Fin : UInt;
   END_VAR
   VAR_OUTPUT
      Mesas_Vacias : Bool;
   END_VAR
   VAR_TEMP
      Aux_contador : UInt;
   END_VAR
BEGIN

REGION Network 1 (SCL)
   FOR #Aux_contador := #Numero_Mesa_Ini TO #Numero_Mesa_Fin DO
       IF "DB900_Estado_Mesas".EstadoVI[#Aux_contador].Etapa_Vacia = false THEN
           #Mesas_Vacias := FALSE;
           RETURN;
       END_IF;
   END_FOR;
   #Mesas_Vacias := true;
END_REGION
END_FUNCTION

FUNCTION "FC502_Actualiza_FIFO_SCR" : Void   // FC502, LAD
{ S7_Optimized_Access := 'FALSE' }
AUTHOR : TLigero
NAME : 20180425
VERSION : 3.1
// stored: AutoNumber false, SetENOAutomatically false
   VAR_INPUT
      DB_FIFO_Ordenes : UInt;
      Num_Scanner : UInt;   // Numero de scanner sobre el que se realiza la busqueda
      Long_FIFO : UInt;
   END_VAR
   VAR_IN_OUT
      FIFO_OK : Bool;
   END_VAR
   VAR_TEMP
      relleno : Byte;
      Indice : Int;
      final : Int;
      retval : Int;
      posicion_actual_N : UInt;
      posicion_siguiente_N1 : UInt;
      Dato_fifo : "ROUT_Orden_Fifo_Scanner";
      Registro_Fifo_vacio : "ROUT_Orden_Fifo_Scanner";
   END_VAR
BEGIN

REGION Network 1 (SCL)
   REGION INICIALIZACIÓN

       #FIFO_OK := FALSE;
       #relleno := 0;
       #retval:= FILL(BVAL := #relleno, BLK => #Registro_Fifo_vacio);
       #posicion_actual_N := 1;
       #final := #Long_FIFO;

   END_REGION
END_REGION

REGION Network 2 (SCL)
   REGION FIFO_1_POS
       //si la fifo es de una posición con borrar esta ya es suficiente.

       IF #Long_FIFO = 1 THEN
           "FC572_Guardar_Datos_Fifo"(DB_FIFO_Ordenes := #DB_FIFO_Ordenes,
                                      Num_Scanner := #Num_Scanner,
                                      Long_FIFO := #Long_FIFO,
                                      Posicion_FIFO := #posicion_actual_N,
                                      Datos_Scanner_Cruce := #Registro_Fifo_vacio);

           #FIFO_OK := true;
           RETURN;

       END_IF;


   END_REGION
END_REGION

REGION Network 3 (SCL)
   REGION FIFO_VARIAS_POSICIONES

       FOR #Indice := 2 TO #final BY 1 DO
           "FC571_Leer_Datos_Fifo"(DB_FIFO_Ordenes:=#DB_FIFO_Ordenes,
                                   Num_Scanner:=#Num_Scanner,
                                   Long_FIFO:=#Long_FIFO,
                                   Posicion_FIFO:=#Indice,
                                   Datos_Scanner_Cruce=>#Dato_fifo);

           "FC572_Guardar_Datos_Fifo"(DB_FIFO_Ordenes:=#DB_FIFO_Ordenes,
                                      Num_Scanner:=#Num_Scanner,
                                      Long_FIFO:=#Long_FIFO,
                                      Posicion_FIFO:=(#Indice-1),
                                      Datos_Scanner_Cruce:=#Dato_fifo);

           "FC572_Guardar_Datos_Fifo"(DB_FIFO_Ordenes := #DB_FIFO_Ordenes,
                                      Num_Scanner := #Num_Scanner,
                                      Long_FIFO := #Long_FIFO,
                                      Posicion_FIFO := #Indice,
                                      Datos_Scanner_Cruce := #Registro_Fifo_vacio);

       END_FOR;
       #FIFO_OK := true;

   END_REGION
END_REGION
END_FUNCTION

FUNCTION "FC509_SIM_Ordenes_SRC_Clasificador_V2" : Void   // FC509, LAD
{ S7_Optimized_Access := 'FALSE' }
AUTHOR : ROUTER
NAME : 20190911
VERSION : 3.1
// NIEVES: 2024/01/29
// Para que en los cruces de más de un destino sea más facil configurar cuantas cajas enviamos por cada cruce, y además hacerlo de la manera más simple para los cruces configurados de manera especial, se configuran en un db las ordenes que queremos que se vayan extrayendo, de manera que podremos decidir en cada momento cuantas enviamos por cada desvío, y la orden que necesitamos para que se ejecute correctamente.
// stored: AutoNumber false, SetENOAutomatically false
   VAR_INPUT
      Numero_cruce : UInt;
      Sacar_orden : Bool;
      Reset : Bool;
   END_VAR
   VAR_OUTPUT
      Orden_FIFO : "ROUT_Orden_Fifo_Scanner";
   END_VAR
   VAR_IN_OUT
      Mem_FP : Bool;
      Aux_contador_cajas : UDInt;
   END_VAR
   VAR_TEMP
      aux_SSCC : DInt;
   END_VAR
   VAR_TEMP   // added for the SCL form of the ladder/FBD networks
      _w1 : Bool;
      _w2 : Bool;
   END_VAR
BEGIN

REGION Network 1: inicializacion
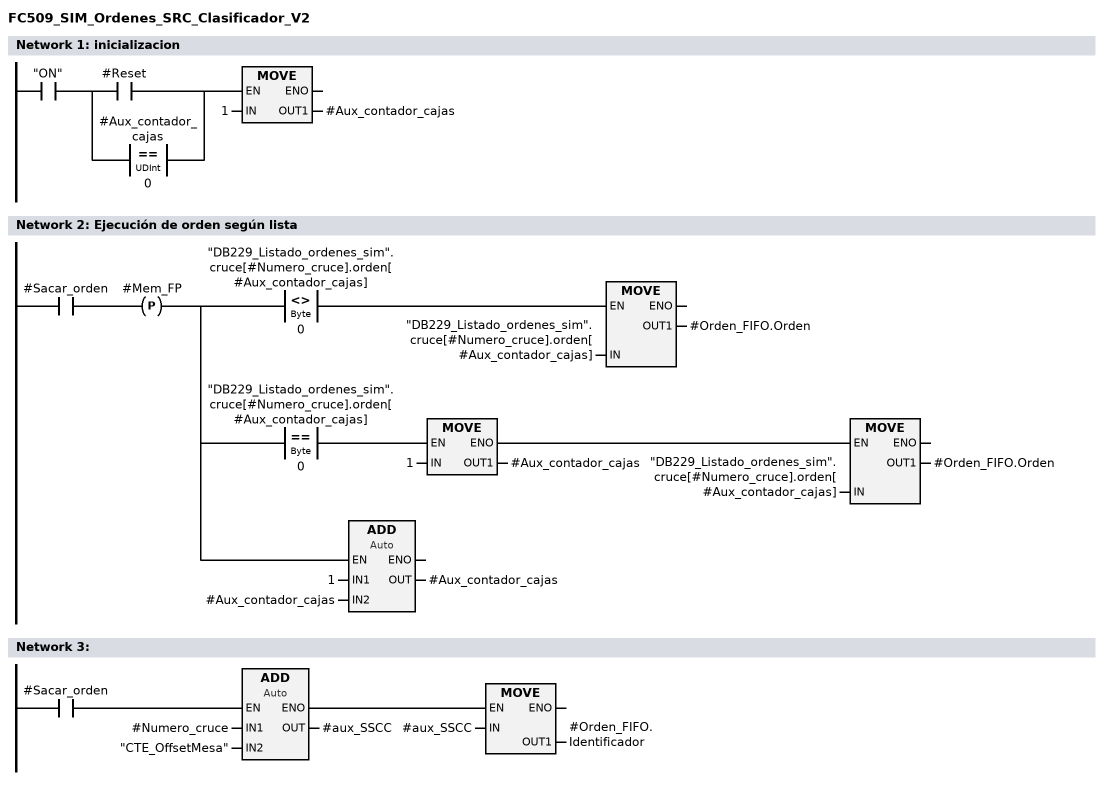
   RUNG wire#powerrail
      Contact( "ON" )
      wire#w1
      Contact( #Reset )
      wire#w2
      Move(in := 1, out1 => #Aux_contador_cajas)
   END_RUNG
   RUNG wire#w1
      { S7_Templates := "SrcType := UDInt" } EQ_Contact(in1 := #Aux_contador_cajas, in2 := 0)
   END_RUNG wire#w2
   // the same network as SCL:
   IF "ON" AND (#Reset OR (#Aux_contador_cajas = 0)) THEN #Aux_contador_cajas := 1; END_IF;
END_REGION

REGION Network 2: Ejecución de orden según lista
   RUNG wire#powerrail
      Contact( #Sacar_orden )
      P_Trig( #Mem_FP )
      wire#w1
      { S7_Templates := "SrcType := Byte" } NE_Contact(in1 := "DB229_Listado_ordenes_sim".cruce[#Numero_cruce].orden[#Aux_contador_cajas], in2 := 0)
      Move(in := "DB229_Listado_ordenes_sim".cruce[#Numero_cruce].orden[#Aux_contador_cajas], out1 => #Orden_FIFO.Orden)
   END_RUNG
   RUNG wire#w1
      { S7_Templates := "SrcType := Byte" } EQ_Contact(in1 := "DB229_Listado_ordenes_sim".cruce[#Numero_cruce].orden[#Aux_contador_cajas], in2 := 0)
      Move(in := 1, out1 => #Aux_contador_cajas)
      Move(in := "DB229_Listado_ordenes_sim".cruce[#Numero_cruce].orden[#Aux_contador_cajas], out1 => #Orden_FIFO.Orden)
   END_RUNG
   RUNG wire#w1
      Add(in1 := 1, in2 := #Aux_contador_cajas, out => #Aux_contador_cajas)
   END_RUNG
   // the same network as SCL:
   #_w1 := #Sacar_orden AND NOT #Mem_FP;   // rising edge
   #Mem_FP := #Sacar_orden;
   IF #_w1 AND ("DB229_Listado_ordenes_sim".cruce[#Numero_cruce].orden[#Aux_contador_cajas] <> 0) THEN
       #Orden_FIFO.Orden := "DB229_Listado_ordenes_sim".cruce[#Numero_cruce].orden[#Aux_contador_cajas];
   END_IF;
   #_w2 := #_w1 AND ("DB229_Listado_ordenes_sim".cruce[#Numero_cruce].orden[#Aux_contador_cajas] = 0);
   IF #_w2 THEN
       #Aux_contador_cajas := 1;
       #Orden_FIFO.Orden := "DB229_Listado_ordenes_sim".cruce[#Numero_cruce].orden[#Aux_contador_cajas];
   END_IF;
   IF #_w1 THEN #Aux_contador_cajas := 1 + #Aux_contador_cajas; END_IF;
END_REGION

REGION Network 3
   RUNG wire#powerrail
      Contact( #Sacar_orden )
      Add(in1 := #Numero_cruce, in2 := "CTE_OffsetMesa", out => #aux_SSCC)
      Move(in := #aux_SSCC, out1 => #Orden_FIFO.Identificador)
   END_RUNG
   // the same network as SCL:
   IF #Sacar_orden THEN
       #aux_SSCC := #Numero_cruce + "CTE_OffsetMesa";
       #Orden_FIFO.Identificador := #aux_SSCC;
   END_IF;
END_REGION
END_FUNCTION

FUNCTION "FC512_TL_EtiquetaLeida_EnMesa_ULINT" : Void   // FC512, LAD
{ S7_Optimized_Access := 'FALSE' }
AUTHOR : T_LIGERO
NAME : 20141014
VERSION : 4.0
// stored: AutoNumber false, SetENOAutomatically false
   VAR_INPUT
      Mesa : UInt;   // Numero de Mesa CON OFFSET
      NumSCR : UInt;   // Numero de Scanner asociada a la mesa
      LongFIFO_SCR : UInt;   // Numero de Lecturas que se pueden Almacenar
      MesaDeJDT02 : Bool;
   END_VAR
   VAR_TEMP
      Datos_scanner : "ROUT_Orden_Fifo_Scanner";
      codigo_string : String[20];
      mesa_string : String[5];
      i : Int;
      FIFO_OK : Bool;
      longitud : Int;
      posicion : Int;
   END_VAR
BEGIN

REGION Network 1 (SCL): escribir los datos en el string
   "FC571_Leer_Datos_Fifo"(DB_FIFO_Ordenes:="ROUT_NDB_FIFO_Odr_SCR",
                           Num_Scanner:=#NumSCR,
                           Long_FIFO:=#LongFIFO_SCR,
                           Posicion_FIFO:=1,
                           Datos_Scanner_Cruce=>#Datos_scanner);

   IF #Datos_scanner.Orden = 0 THEN
       RETURN;
   END_IF;




   // MIRAR SI TENEMOS ESPACIO PARA EMITIR EL MENSAJE ANTES DE FORMATEARLO
   IF #MesaDeJDT02 = true THEN
       REGION buscar en JDT2

           #posicion := -1;
           FOR #i := 0 TO 100 BY 1 DO
               #longitud := LEN("DB197_eventos_generados_routing_JDT2".evento[#i]);
               IF #longitud = 0 THEN
                   #posicion := #i;
                   EXIT;
               END_IF;
           END_FOR;

           // si no hay sitio para escribir salimos del bloque
           IF #posicion = -1 THEN
               RETURN;
           END_IF;
       END_REGION
       ;
   ELSE
       REGION buscar en JDT1

           #posicion := -1;
           FOR #i := 0 TO 100 BY 1 DO
               #longitud := LEN("DB198_eventos_generados_routing_JDT1".evento[#i]);
               IF #longitud = 0 THEN
                   #posicion := #i;
                   EXIT;
               END_IF;
           END_FOR;

           // si no hay sitio para escribir salimos del bloque
           IF #posicion = -1 THEN
               RETURN;
           END_IF;
       END_REGION
   END_IF;
   // buscamos hueco en el db donde vamos a escribir los eventos antes de empezar la conversión
   // 

   // si hay sitio para convertir iniciamos la conversión de los parametros a enviar en el mensaje

   #mesa_string :=  DELETE(IN := (UINT_TO_STRING(IN := #Mesa)), L := 1, P := 1);
   #codigo_string := DELETE(IN := (ULINT_TO_STRING(IN := #Datos_scanner.Identificador)), L := 1, P := 1);

   // concatenamos el mensaje 
   // 
   IF #MesaDeJDT02 = true THEN

       "DB197_eventos_generados_routing_JDT2".evento[#posicion] := CONCAT(IN1 := '{PRES[MESA]', IN2 := #mesa_string, IN3 := '[SSCC]', IN4 := #codigo_string, IN5 := '[MOTI]NORM', IN6 :="DB921_DATOS_FECHA_HORA".TIME_STAMP , IN7:='}');

       ELSE
           "DB198_eventos_generados_routing_JDT1".evento[#posicion] := CONCAT(IN1 := '{PRES[MESA]', IN2 := #mesa_string, IN3 := '[SSCC]', IN4 := #codigo_string, IN5 := '[MOTI]NORM', IN6 :="DB921_DATOS_FECHA_HORA".TIME_STAMP , IN7:='}');

   END_IF;

       "FC502_Actualiza_FIFO_SCR"(DB_FIFO_Ordenes:="ROUT_NDB_FIFO_Odr_SCR",
                                  Num_Scanner:=#NumSCR,
                                  Long_FIFO:=#LongFIFO_SCR,
                                  FIFO_OK:=#FIFO_OK);
END_REGION
END_FUNCTION

FUNCTION "FC513_TL_Etiqueta_EnMesaCruce_ULINT" : Void   // FC513, LAD
{ S7_Optimized_Access := 'FALSE' }
// stored: AutoNumber false, SetENOAutomatically false
   VAR_INPUT
      Mesa : UInt;   // Numero de Mesa CON OFFSET
      Mesa_S01 : UInt;   // Mesa de Salida por S01 CON OFFSET
      Mesa_S02 : UInt;   // Mesa de Salida por S02 CON OFFSET
      Mesa_S03 : UInt;   // Mesa de Salida por S03 CON OFFSET
      Mesa_S04 : UInt;   // Mesa de Salida por S04 CON OFFSET
      Etiqueta : ULInt;   // Etiqueta
      OrdenEjecutada : UInt;   // Orden Ejecutada en el Cruce
      MesaDeJDT02 : Bool;
   END_VAR
   VAR_TEMP
      MesaTMP : UDInt;
      MotivoTMP : UDInt;
      Posicion : Int;
      i : Int;
      longitud : Int;
      string_motivo : String[10];
      string_mesa : String[12];
      codigo_string : String[20];
   END_VAR
BEGIN

REGION Network 1 (SCL)
   //---------------------------------------------------------------------------------------------
   // --- 
   // --- Condiciones para enviar el Nuevo Evento
   // ---     Cerrado el Protocolo de la Mesa
   // --- Recoger - Presencias de la Mesa
   // --- Emitiendo Mensajes
   // ---
   // ---------------------------------------------------------------------------------------------
   // ------- Cerrado el Protocolo de la Mesa
   // 
   IF "DB810_ColasMesas".Colas[#Mesa].EstadoPresenciaMesa <> 0 THEN
       RETURN;
   END_IF;


   // ---------------------------------------------------------------------------------------------
   // ------- Recoger - Presencias de la Mesa
   // ---------------------------------------------------------------------------------------------

   IF "DB840_Emision".Mesa[#Mesa].Protocolo.PresRouter = FALSE THEN
       RETURN;
   END_IF;

   // ---------------------------------------------------------------------------------------------
   // ------- Recoger Datos para la Generacion del Evento

   #MotivoTMP := #OrdenEjecutada / 10;
   #MesaTMP := #OrdenEjecutada MOD 10;
END_REGION

REGION Network 2 (SCL)
   // miramos si tenemos hueco para emitir hacia el jdt que nos corresponde
   // 
   IF #MesaDeJDT02=true THEN
       REGION buscar en JDT2

           #Posicion := -1;
           FOR #i := 0 TO 100 BY 1 DO
               #longitud := LEN("DB197_eventos_generados_routing_JDT2".evento[#i]);
               IF #longitud = 0 THEN
                   #Posicion := #i;
                   EXIT;
               END_IF;
           END_FOR;

           // si no hay sitio para escribir salimos del bloque
           IF #Posicion = -1 THEN
               RETURN;
           END_IF;
       END_REGION
       ;
   ELSE
       REGION buscar en JDT1

           #Posicion := -1;
           FOR #i := 0 TO 100 BY 1 DO
               #longitud := LEN("DB198_eventos_generados_routing_JDT1".evento[#i]);
               IF #longitud = 0 THEN
                   #Posicion := #i;
                   EXIT;
               END_IF;
           END_FOR;

           // si no hay sitio para escribir salimos del bloque
           IF #Posicion = -1 THEN
               RETURN;
           END_IF;
       END_REGION
   END_IF;
END_REGION

REGION Network 3 (SCL)

   CASE #MotivoTMP OF
       0:
           #string_motivo := '[MOTI]NORM';         // --- Escribir - Motivo NORMAL  (0)
       1:
           #string_motivo := '[MOTI]BLOQ';     // --- Escribir - Motivo BLOQUEO (1)
       2:
           #string_motivo := '[MOTI]VACI';   // --- Escribir - Motivo VACIADO (2)
       3:
           #string_motivo := '[MOTI]ERRO';  // --- Escribir - Motivo ETIQUETA ERROR (3)
       4:
           #string_motivo := '[MOTI]NENC';// --- Escribir - Motivo ETIQUETA NO ENCONTRADA (4)
       5:
           #string_motivo := '[MOTI]INIC'; // --- Escribir - Motivo Ejecucion por INICIALIZACION (5)
       6:
           #string_motivo := '[MOTI]XJDT';// --- Escribir - Motivo Ejecucion por JDT (6)
       7:
           #string_motivo := '[MOTI]BLKC';  // --- Escribir - Motivo Ejecucion por Bloqueo intentando Continuar (7)
       8:
           #string_motivo := '[MOTI]BLKE'; // --- Escribir - Motivo Ejecucion por Bloqueo intentando Entrar (8)


       ELSE
           #string_motivo := '[MOTI]DESC';

   END_CASE;

   CASE #MesaTMP OF

       1:
           #string_mesa := CONCAT(IN1 := '[MESA]', IN2 := DELETE(IN := (UDINT_TO_STRING(IN := #Mesa_S01)), L := 1, P := 1));
       2:
           #string_mesa := CONCAT(IN1 := '[MESA]', IN2 := DELETE(IN := (UDINT_TO_STRING(IN := #Mesa_S02)), L := 1, P := 1));
       3:
           #string_mesa := CONCAT(IN1 := '[MESA]', IN2 := DELETE(IN := (UDINT_TO_STRING(IN := #Mesa_S03)), L := 1, P := 1));
       4:
           #string_mesa := CONCAT(IN1 := '[MESA]', IN2 := DELETE(IN := (UDINT_TO_STRING(IN := #Mesa_S04 )), L := 1, P := 1));

       ELSE  // Statement section ELSE
           #string_mesa := CONCAT(IN1 := '[MESA]', IN2 := DELETE(IN := (UDINT_TO_STRING(IN := #Mesa)), L := 1, P := 1));

   END_CASE;

   #codigo_string := DELETE(IN := (ULINT_TO_STRING(IN :=#Etiqueta)), L := 1, P := 1);


   IF #MesaDeJDT02 = true THEN

       "DB197_eventos_generados_routing_JDT2".evento[#Posicion] := CONCAT(IN1 := '{PRES', IN2 := #string_mesa, IN3 := '[SSCC]', IN4 := #codigo_string, IN5 := #string_motivo, IN6 := "DB921_DATOS_FECHA_HORA".TIME_STAMP, IN7:='}');

   ELSE
       "DB198_eventos_generados_routing_JDT1".evento[#Posicion] := CONCAT(IN1 := '{PRES', IN2 := #string_mesa, IN3 := '[SSCC]', IN4 := #codigo_string, IN5 := #string_motivo, IN6 := "DB921_DATOS_FECHA_HORA".TIME_STAMP, IN7:='}');

   END_IF;

   "DB841_Recepcion".Mesa[#Mesa].Protocolo.EmiOK := TRUE;
   "DB810_ColasMesas".Colas[#Mesa].EstadoPresenciaMesa := 1;
END_REGION
END_FUNCTION

FUNCTION "FC521_Re_Evalua_Etiqueta_Ulint" : Void   // FC521, SCL
{ S7_Optimized_Access := 'FALSE' }
// stored: AutoNumber false, SetENOAutomatically false
   VAR_INPUT
      Num_Scanner_Entrada : UInt;   // Numero de scanner sobre el que se realiza la busqueda
      DB_FIFO_Ordenes_Entrada : UInt;
      Long_Fifo_Entrada : UInt;
      Num_Scanner_Salida : UInt;
      DB_FIFO_Orden_Salida : UInt;
      Long_fifo_Salida : UInt;
   END_VAR
   VAR_TEMP
      Datos_scanner_reevaluar : "ROUT_Orden_Fifo_Scanner";
      Cola : UDInt;
      Posicion_Etiqueta_TMP : UInt;
      Num_Inic : UInt;
      Tipo_SCR : UInt;
      Etiqueta : ULInt;
      primer_bit : UInt;
      numero_bits : UInt;
      contador : UInt;
      cont_aux : UInt;
      orden : Byte;
      orden_aux AT orden : Array[0..7] of Bool;
      Inic_bits : Array[1..8] of Bool;
      Reg_Etiq_Temp : "ROUT_Reg_Etiqueta";
      Datos_fifo : "ROUT_Orden_Fifo_Scanner";
      Datos_fifo_tmp : "ROUT_Orden_Fifo_Scanner";
      Numero_SCR : UInt;
      posicion_fifo : UInt;
      fifo_ok : Bool;
   END_VAR
BEGIN
   REGION buscar_datos_reevaluar
       "FC571_Leer_Datos_Fifo"(DB_FIFO_Ordenes := #DB_FIFO_Ordenes_Entrada,
                               Num_Scanner := #Num_Scanner_Entrada,
                               Long_FIFO := #Long_Fifo_Entrada,
                               Posicion_FIFO := 1,
                               Datos_Scanner_Cruce => #Datos_scanner_reevaluar);

       IF #Datos_scanner_reevaluar.Orden = 0 THEN
           RETURN;
       END_IF;

   END_REGION

   REGION inicilizar

       #Etiqueta := #Datos_scanner_reevaluar.Identificador;
       #Posicion_Etiqueta_TMP := 0;
       #Num_Inic := "DB912_Tipo_Scanner_Router".SCANNER[#Num_Scanner_Salida].Num_Inicializacion;
       #Tipo_SCR := "DB912_Tipo_Scanner_Router".SCANNER[#Num_Scanner_Salida].Tipo;
       #Numero_SCR := #Num_Scanner_Salida;
       #Datos_fifo.Identificador := 0;
       #Datos_fifo.Libre := 0;
       #Datos_fifo.Orden := 0;
       SCATTER(IN := "Estado_inicializacion",
               OUT => #Inic_bits);

   END_REGION
   // si seguimos es porque tenemos una etiqueta que tiene que ser re-evaluada

   REGION comprobar_inicializacion
       // comprobamos si el scanner que estamos comprobando está en proceso de inicialización
       IF ((#Num_Inic >= 1) AND (#Num_Inic <= 8)) THEN
           // si tiene un numero de inicialización configurado, comprobamos si está activo
           IF (#Inic_bits[#Num_Inic] = true) THEN
               GOTO proceso_INIC;
           END_IF;
       END_IF;

   END_REGION

   REGION comprobar_etiqueta

       IF #Etiqueta <= 0 THEN
           GOTO error_lectura;
       ELSE
           #Cola := #Etiqueta MOD "ROUT_N_Colas";        // calculamos el numero de cola
       END_IF;
   END_REGION

   #Posicion_Etiqueta_TMP := "DB212_Cola_Activa".Cola[#Cola];

   // comprobamos si existe alguna etiqueta en esa cola

   elegir_db_busqueda:

   // si esa etiqueta no está dada de alta en las colas es que no está activa 
   IF #Posicion_Etiqueta_TMP = 0 THEN
       GOTO lectura_NENC;
   END_IF;


   REGION elegir_db_busqueda
       CASE #Posicion_Etiqueta_TMP OF
           1..1000:
               GOTO busca_1_999;
           1001..2000:
               GOTO busca_1k;
           2001..3000:
               GOTO busca_2k;
           3001..4000:
               GOTO busca_3k;
           ELSE

               GOTO lectura_NENC;
       END_CASE;
   END_REGION

   ////////////////////////////////////////////
   REGION busca_1_a_1000
   busca_1_999:
       IF #Etiqueta = "DB201_RegEtiquetas_0001_1000".Reg_Etiqueta[#Posicion_Etiqueta_TMP].CDB THEN
           #Reg_Etiq_Temp := "DB201_RegEtiquetas_0001_1000".Reg_Etiqueta[#Posicion_Etiqueta_TMP];
           GOTO lectura_encontrada;
       ELSE
           #Posicion_Etiqueta_TMP := "DB201_RegEtiquetas_0001_1000".Reg_Etiqueta[#Posicion_Etiqueta_TMP].Posterior;
           GOTO elegir_db_busqueda;
       END_IF;
   END_REGION

   ////////////////////////////////////////////
   REGION busca_1001_a_2000
   busca_1k:
       #Posicion_Etiqueta_TMP := #Posicion_Etiqueta_TMP - 1000;
       IF #Etiqueta = "DB202_RegEtiquetas_1001_2000".Reg_Etiqueta[#Posicion_Etiqueta_TMP].CDB THEN
           #Reg_Etiq_Temp := "DB202_RegEtiquetas_1001_2000".Reg_Etiqueta[#Posicion_Etiqueta_TMP];
           GOTO lectura_encontrada;
       ELSE
           #Posicion_Etiqueta_TMP := "DB202_RegEtiquetas_1001_2000".Reg_Etiqueta[#Posicion_Etiqueta_TMP].Posterior;
           GOTO elegir_db_busqueda;
       END_IF;
   END_REGION

   ////////////////////////////////////////////
   REGION busca_2001_a_3000
   busca_2k:
       #Posicion_Etiqueta_TMP := #Posicion_Etiqueta_TMP - 2000;
       IF #Etiqueta = "DB203_RegEtiquetas_2001_3000".Reg_Etiqueta[#Posicion_Etiqueta_TMP].CDB THEN
           #Reg_Etiq_Temp := "DB203_RegEtiquetas_2001_3000".Reg_Etiqueta[#Posicion_Etiqueta_TMP];
           GOTO lectura_encontrada;
       ELSE
           #Posicion_Etiqueta_TMP := "DB203_RegEtiquetas_2001_3000".Reg_Etiqueta[#Posicion_Etiqueta_TMP].Posterior;
           GOTO elegir_db_busqueda;
       END_IF;

   END_REGION

   ////////////////////////////////////////////
   REGION busca_3001_a_4000
   busca_3k:
       #Posicion_Etiqueta_TMP := #Posicion_Etiqueta_TMP - 3000;
       IF #Etiqueta = "DB204_RegEtiquetas_3001_4000".Reg_Etiqueta[#Posicion_Etiqueta_TMP].CDB THEN
           #Reg_Etiq_Temp := "DB204_RegEtiquetas_3001_4000".Reg_Etiqueta[#Posicion_Etiqueta_TMP];
           GOTO lectura_encontrada;
       ELSE
           #Posicion_Etiqueta_TMP := "DB204_RegEtiquetas_3001_4000".Reg_Etiqueta[#Posicion_Etiqueta_TMP].Posterior;
           GOTO elegir_db_busqueda;
       END_IF
       ;
   END_REGION

   REGION Especial_error_lectura
   error_lectura:
       #Reg_Etiq_Temp := "DB209_Reg_Etquetas_Esp_Activa".Reg_Etiqueta[1];
       #Datos_fifo.Orden := w#16#90;
       IF #Tipo_SCR = 2 THEN // tipo validación
           #Datos_fifo.Identificador := #Etiqueta;
           GOTO guardar_orden;
       END_IF;
       GOTO extraer_orden;
   END_REGION
   REGION Especial_NENC
   lectura_NENC:
       #Datos_fifo.Identificador := #Etiqueta;
       IF (#Tipo_SCR = 2) THEN
           #Datos_fifo.Orden := w#16#80;

           GOTO guardar_orden;
       END_IF;
       #Reg_Etiq_Temp := "DB209_Reg_Etquetas_Esp_Activa".Reg_Etiqueta[2];
       #Datos_fifo.Orden := w#16#A0;
       // hay dos casos posibles. si el escanner es normal extrae orden normal
       // si es de validacion de etiqueta, extrae el predeterminado
       GOTO extraer_orden;
   END_REGION
   REGION Especial_INIC
   proceso_INIC:
       #Reg_Etiq_Temp := "DB209_Reg_Etquetas_Esp_Activa".Reg_Etiqueta[3];
       #Datos_fifo.Orden := w#16#C0;
       GOTO extraer_orden;
   END_REGION
   REGION lectura_ok
   lectura_encontrada:
       #Datos_fifo.Identificador := #Etiqueta;
       IF #Tipo_SCR = 2 THEN
           #Datos_fifo.Orden := w#16#81;
           GOTO guardar_orden;
       ELSE
           #Datos_fifo.Orden := w#16#80;
           GOTO extraer_orden;
       END_IF;


   END_REGION

   REGION Extraer orden
   extraer_orden:
       #Datos_fifo.Identificador := #Etiqueta;
       // proceso extracción de la orden
       // miramos cual es el primer bit que tenemos que sacar de la orden
       #primer_bit := "DB912_Tipo_Scanner_Router".SCANNER[#Numero_SCR].Bit_Ini_Ordenes;
       #numero_bits := "DB912_Tipo_Scanner_Router".SCANNER[#Numero_SCR].N_Bits_Orden;
       #cont_aux := 0;
       #orden :=#Datos_fifo.Orden;
       FOR #contador := #primer_bit TO (#primer_bit + #numero_bits - 1) DO
           #orden_aux[#cont_aux] := #Reg_Etiq_Temp.BIT_Orden[#contador];
           #cont_aux += 1;
       END_FOR;
       #Datos_fifo.Orden :=#orden;
       ;
   END_REGION

   REGION Guardar_Orden

   guardar_orden:
       // miramos si ya hay algo en la fifo
       // como puede tener cualquier tamaño, tenemos que buscar la siguiente posición libre
       // para encolar la orden
       // 



       FOR #posicion_fifo:=1 TO #Long_fifo_Salida BY 1 DO

           "FC571_Leer_Datos_Fifo"(DB_FIFO_Ordenes :=  #DB_FIFO_Orden_Salida,
                               Num_Scanner := #Numero_SCR,
                               Long_FIFO := #Long_fifo_Salida,
                               Posicion_FIFO := #posicion_fifo,
                               Datos_Scanner_Cruce => #Datos_fifo_tmp);
       // comprobamos si la posición está ocupada
       // 
       IF #Datos_fifo_tmp.Orden = 0 THEN
           // volcamos los datos actualizados
           "FC572_Guardar_Datos_Fifo"(DB_FIFO_Ordenes := #DB_FIFO_Orden_Salida,
                                      Num_Scanner := #Numero_SCR,
                                      Long_FIFO :=  #Long_fifo_Salida,
                                      Posicion_FIFO := #posicion_fifo,
                                      Datos_Scanner_Cruce := #Datos_fifo);
           // borramos de la fifo de entrada el dato que ya hemos re-evaluado
           // 
   "FC502_Actualiza_FIFO_SCR"(DB_FIFO_Ordenes:=#DB_FIFO_Ordenes_Entrada,
                              Num_Scanner:=#Num_Scanner_Entrada,
                              Long_FIFO:=#Long_Fifo_Entrada,
                              FIFO_OK:=#fifo_ok);


           RETURN;
       END_IF;

   END_FOR;

   // si no hemos encontrado ninguna posición libre en la fifo, generamos un vaciado en la primera posición

           #Datos_fifo.Orden := w#16#FF;
           "FC572_Guardar_Datos_Fifo"(DB_FIFO_Ordenes := #DB_FIFO_Orden_Salida,
                                      Num_Scanner := #Numero_SCR,
                                      Long_FIFO := #Long_fifo_Salida,
                                      Posicion_FIFO := 1,
                                      Datos_Scanner_Cruce := #Datos_fifo);

           // borramos de la fifo de entrada el dato que ya hemos re-evaluado   
           "FC502_Actualiza_FIFO_SCR"(DB_FIFO_Ordenes := #DB_FIFO_Ordenes_Entrada,
                                      Num_Scanner := #Num_Scanner_Entrada,
                                      Long_FIFO := #Long_Fifo_Entrada,
                                      FIFO_OK := #fifo_ok);




   END_REGION
END_FUNCTION

FUNCTION "FC532_Estado_Ocupacion" : Void   // FC532, STL
{ S7_Optimized_Access := 'FALSE' }
AUTHOR : ROUTER
NAME : 20130631
VERSION : 3.1
// stored: AutoNumber false
   VAR_INPUT
      NumeroMesa : UInt;   // Numero de Mesa
      EstadoMesaVacia : Bool;   // Vacia=1
      MesaDeJDT02 : Bool;
   END_VAR
   VAR_IN_OUT
      MemEstadoOcupa : Byte;
   END_VAR
   VAR_TEMP
      DBEventos : Word;   // Numero del DB de Eventos
      NumBytes : UInt;   // Numero de Bytes existentes en el DB de Eventos
      PunteroEventos : DWord;   // Puntero al DB de Eventos
      ValorTMP : UDInt;
      OffsetTMP : UInt;
      NumDBEventos : UInt;
      MaxBytes : UInt;
   END_VAR
BEGIN

NETWORK
TITLE = 
// ---------------------------------------------------------------------
// --- Mirar si estamos activos para mandar el estado de la mesa

      SET;
      A     "DB902_Estado_ZonaMesa".EstadoMesas[#NumeroMesa].Marcha_CBx;  //#Estado_Zona_Mesa.Marcha_CBx
      JC    Continua;

      L     0;
      T     #MemEstadoOcupa;

      JU    Fin_funcion;



NETWORK
TITLE = Acciones
// ---------------------------------------------------------------------
// --- Mirar el Estado de Ocupacion de la Mesa (Si ha Cambiado)

Continua:SET;  // Mirar si ha cambiado de Estado
      A     #EstadoMesaVacia;  // Estado diferente
      A(;
      O(;
      L     #MemEstadoOcupa;
      L     2;
      ==I;
      );
      O(;
      L     #MemEstadoOcupa;
      L     0;
      ==I;
      );
      );
      JC    Emitir_estado;

      SET;
      AN    #EstadoMesaVacia;
      A(;
      O(;
      L     #MemEstadoOcupa;
      L     1;
      ==I;
      );
      O(;
      L     #MemEstadoOcupa;
      L     0;
      ==I;
      );
      );
      JC    Emitir_estado;

      JU    Fin_funcion;  // No ha Cambiado de Estado


NETWORK
TITLE = Evento de Estado de Ocupacion de la Mesa
// ---------------------------------------------------------------------
// ---
// ---
// ---   Pasos a Seguir para el Formateo del Evento
// ---
// ---   * Mirar si hay sitio para generar el nuevo evento
// ---       * Inicializo NumBytes y Puntero al DB de Eventos Generados
// ---       * Calcula el tamaño de bytes que hay en el DB de Eventos Generados
// ---       * Comprobar si hay sitio para un evento más
// ---   *  Formatear el Evento
// ---
// ---
// ---------------------------------------------------------------------


// ---------------------------------------------------------------------
// --- Mirar si hay sitio para generar un evento más

Emitir_estado:SET;
      L     "JDT1_NDB_EventosEmi";
      T     #DBEventos;
      T     #NumDBEventos;
      L     "JDT1_MaxBytes";
      T     #MaxBytes;

// ---------------------------------------------------------------------
/// Inicio --> Pertenece al JDT 02

      AN    #MesaDeJDT02;
      JC    No_es_JdT02;

      L     "JDT2_NDB_EventosEmi";
      T     #DBEventos;
      T     #NumDBEventos;
      L     "JDT2_MaxBytes";
      T     #MaxBytes;

No_es_JdT02:NOP   0;

/// Final --> Pertenece al JDT 02
// ---------------------------------------------------------------------


      L     0;
      T     #NumBytes;  // Inicializo el numero de Bytes
      T     #PunteroEventos;  // Inicializo el puntero de Eventos Generados


Buscar_hueco:SET;
      OPN   DB [#DBEventos];  // Calcula el tamaño de bytes que hay en el DB
      L     DBB [#PunteroEventos];
      L     0;
      ==I;
      JC    Valida_hueco;  // Buscamos el final del DB = 0

      OPN   DB [#DBEventos];
      L     DBB [#PunteroEventos];
      L     ' ';
      ==I;
      JC    Valida_hueco;  // Buscamos el final del DB = ' '

      L     #PunteroEventos;  // Incremento de P#1.0
      L     P#1.0;
      +D;
      T     #PunteroEventos;

      JU    Buscar_hueco;  // Continuar con el siguiente posicion


Valida_hueco:SET;
      L     #PunteroEventos;  // Sacamos el NumBytes Escritos
      SRD   3;
      T     #NumBytes;

      L     #NumBytes;  // Miramos si hay sitio
      L     #MaxBytes;  // Max. que se pueden emitir, parametro
      >I;
      JC    Fin_funcion;  // No se pueden generar más eventos

// ---------------------------------------------------------------------
// --- Formatear el evento de Estado de Ocupacion de la Mesa

      L     #PunteroEventos;
      LAR2;  // Puntero al DB de Eventos Generados

      TAR2;  // Mirar si es el primer evento de la lista
      L     0;
      ==I;
      JC    Primer_evento;  // Es el primero

      OPN   DB [#DBEventos];
      L     ',';  // Separador entre eventos ','
      T     DBB [AR2, P#0.0];
      +AR2  P#1.0;


Primer_evento:SET;
      OPN   DB [#DBEventos];  // DB de Eventos Generados (A Emitir)
      L     '{';  // Inicio de Evento '{'
      T     DBB [AR2, P#0.0];
      +AR2  P#1.0;

      L     'DIDA';  // --- Evento 'DIDA'
      T     DBD [AR2, P#0.0];
      +AR2  P#4.0;

      OPN   DB [#DBEventos];
      L     '[';  // --- Evento - Atributo Tipo '[TIPO]'
      T     DBB [AR2, P#0.0];
      L     'TIPO';
      T     DBD [AR2, P#1.0];
      L     ']';
      T     DBB [AR2, P#5.0];
      +AR2  P#6.0;

      OPN   DB [#DBEventos];
      L     'MESA';  // Tipo Llave 'MESA'
      T     DBD [AR2, P#0.0];
      +AR2  P#4.0;

      L     '[';  // --- Evento - Atributo Numero de Mesa '[NUME]'
      T     DBB [AR2, P#0.0];
      L     'NUME';
      T     DBD [AR2, P#1.0];
      L     ']';
      T     DBB [AR2, P#5.0];
      +AR2  P#6.0;

      L     "CTE_OffsetMesa";
      L     #NumeroMesa;  // Numero de la Llave
      +I;
      T     #ValorTMP;

// --- Convertir Valor a ASCII

      TAR2;
      SRD   3;
      T     #NumBytes;  // Miro que offset tiene la String

      CALL  "FC893_Obtener_StringDelAtributo"
      ( DB_String := #NumDBEventos,
        OffsetIni := #NumBytes,
        Valor     := #ValorTMP,
        OffsetFin := #OffsetTMP
      );  // Llamo a ObtenerStrinAtributo

      L     #OffsetTMP;
      SLD   3;
      LAR2;  // Recupero que offset tiene la String

// --- Ya esta convertido el Valor a ASCII

      OPN   DB [#DBEventos];
      L     '[';  // --- Evento - Atributo de Estado '[FULL]'
      T     DBB [AR2, P#0.0];
      L     'FULL';
      T     DBD [AR2, P#1.0];
      L     ']';
      T     DBB [AR2, P#5.0];
      +AR2  P#6.0;

      L     'VACI';
      SET;
      A     #EstadoMesaVacia;
      JC    _EST;

      L     'LLEN';

_EST: OPN   DB [#DBEventos];
      T     DBD [AR2, P#0.0];
      +AR2  P#4.0;

      OPN   DB [#DBEventos];  // DB de Eventos Generados (A Emitir)
      L     '}';  // --- Fin de Evento '}'
      T     DBB [AR2, P#0.0];
      +AR2  P#1.0;

// ---------------------------------------------------------------------
// --- Final del Evento

      SET;
      A     #EstadoMesaVacia;
      JCN   VACI;
      L     DINT#1;
      T     #MemEstadoOcupa;

VACI: SET;
      AN    #EstadoMesaVacia;
      JCN   Fin_funcion;

      L     DINT#2;
      T     #MemEstadoOcupa;

      JU    Fin_funcion;  //Final del Formateo del Elento


NETWORK
TITLE = Final de la Funcion
// ---------------------------------------------------------------------
// --- Final de la Funcion

Fin_funcion:NOP   0;

END_FUNCTION

FUNCTION "FC572_Guardar_Datos_Fifo" : Void   // FC572, STL
{ S7_Optimized_Access := 'FALSE' }
// stored: AutoNumber false
   VAR_INPUT
      DB_FIFO_Ordenes : UInt;
      Num_Scanner : UInt;   // Numero de scanner sobre el que se realiza la busqueda
      Long_FIFO : UInt;
      Posicion_FIFO : UInt;
      Datos_Scanner_Cruce : "ROUT_Orden_Fifo_Scanner";
   END_VAR
   VAR_TEMP
      Guardar_AR2 : DWord;
      P_Inicio_Datos : DWord;
      P_Any_Datos : Any;
      NumDB : Word;
      MaxRegistros : UInt;
      LongRegistro : UInt;
      OffsetPrimerRegistro : UInt;
      ValorReturn : Int;
      Elementos_X_Registro : Int;
      Relleno : Byte;
   END_VAR
BEGIN

NETWORK
TITLE = Inicializar Variables
//////////////////////////////////////////////////////////////////////////
/// - Datos del DB a leer

      L     #DB_FIFO_Ordenes;  // - Numero de DB a Leer
      T     #NumDB;
      L     "CTE_MaxMesas";  // - Numero Maximo de Registros
      T     #MaxRegistros;
      L     "ROUT_Long_Reg_Datos_FIFO";  // - Longitud de la estructura del Registro
      T     #LongRegistro;
      L     #Long_FIFO;
      T     #Elementos_X_Registro;
      L     0;  // - Offset del Primer Registro
      T     #OffsetPrimerRegistro;


//////////////////////////////////////////////////////////////////////////


NETWORK
TITLE = Posicionarse en el Registro
//////////////////////////////////////////////////////////////////////////
/// - Comprobar si el registro existe (Maximo de Registros)

      L     #Num_Scanner;
      L     #MaxRegistros;
      >I;
      JC    Error_MaxRegistros;


//////////////////////////////////////////////////////////////////////////
/// - Calculo de la posicion del registro

      L     #Num_Scanner;
      L     #LongRegistro;
      *I;
      L     #Elementos_X_Registro;
      *I;
      L     #OffsetPrimerRegistro;
      +I;
      SLD   3;
      T     #P_Inicio_Datos;


// miramos si tenemos que sacar un registro diferente del primero

      L     #Posicion_FIFO;
      L     1;
      ==I;
      JC    guardar_datos;
// si es un registro diferente del primero, calculamos el offset para colocarnos en el registro correcto

      L     #Posicion_FIFO;
      L     1;
      -I;
      L     #LongRegistro;
      *I;
      SLD   3;
      L     #P_Inicio_Datos;
      +D;
      T     #P_Inicio_Datos;



NETWORK
TITLE = Transferenica del Registro
//////////////////////////////////////////////////////////////////////////
/// - Calculo del Puntero Any de los Datos
guardar_datos:NOP   0;
      TAR2  #Guardar_AR2;  // - Guardar el Puntero AR2

      LAR2  P##P_Any_Datos;  // - Direccion del Puntero Any
      L     B#16#10;  //   10H para S7
      T     LB [AR2, P#0.0];
      L     B#16#2;  //   Tipo de Datos (BYTE)
      T     LB [AR2, P#1.0];
      L     #LongRegistro;  //   Longitud de la Estructura
      T     LW [AR2, P#2.0];
      L     #NumDB;  //   Numero de DB
      T     LW [AR2, P#4.0];
      L     #P_Inicio_Datos;  //   Direccion de Inicio
      T     LD [AR2, P#6.0];
      L     B#16#84;  //   El Area de Memoria = DB
      T     LB [AR2, P#6.0];

      LAR2  #Guardar_AR2;  // - Recuperar el Puntero AR2

//////////////////////////////////////////////////////////////////////////
/// - Transferencia de los Datos a Leer

      CALL  BLKMOV
      ( SRCBLK  := #Datos_Scanner_Cruce,
        RET_VAL := #ValorReturn,
        DSTBLK  := #P_Any_Datos
      );

      L     #ValorReturn;  // - Comprobar que se ha leido el registro
      L     0;
      <>I;
      JC    Error_LecturaDelRegisto;


//////////////////////////////////////////////////////////////////////////
/// - Fin de la Lectura del Registro

      BE;  // - Finalizar bloque



NETWORK
TITLE = Errores en el Sistema de Lectura
//////////////////////////////////////////////////////////////////////////
/// - Numero De Maximo de Registros Sobrepasado

Error_MaxRegistros:NOP   0;
      BE;  // - Finalizar bloque

////////////////////////////////////////////////////
/// - Error a Leer el Registro

Error_LecturaDelRegisto:NOP   0;
      BE;  // - Finalizar bloque


END_FUNCTION

FUNCTION "FC716_Router_BuscarEtiqueta_Lint_y_sacar_orden" : Void   // FC716, SCL
{ S7_Optimized_Access := 'FALSE' }
// stored: AutoNumber false, SetENOAutomatically false
   VAR_INPUT
      Etiqueta : ULInt;   // Etiqueta A Buscar en la Base de Datos
      Numero_SCR : UInt;
   END_VAR
   VAR_TEMP
      Cola : UDInt;
      EtiquetaTMP : ULInt;
      Posicion_Etiqueta_TMP : UInt;
      aux_pos : UInt;
      Num_Inic : UInt;
      Tipo_SCR : UInt;
      primer_bit : UInt;
      numero_bits : UInt;
      contador : UInt;
      CERO : Byte;
      Retval : Int;
      orden : Byte;
      orden_aux AT orden : Array[0..7] of Bool;
      cont_aux : UInt;
      Inic_bits : Array[1..8] of Bool;
      Reg_Etiq_Temp : "ROUT_Reg_Etiqueta";
      Datos_fifo : "ROUT_Orden_Fifo_Scanner";
      datos_actuales_fifo : "ROUT_Orden_Fifo_Scanner";
   END_VAR
BEGIN
   REGION inicilizar

       #EtiquetaTMP := #Etiqueta;
       #Posicion_Etiqueta_TMP := 0;
       #CERO := 0;
       #Num_Inic := "DB912_Tipo_Scanner_Router".SCANNER[#Numero_SCR].Num_Inicializacion;
       #Tipo_SCR := "DB912_Tipo_Scanner_Router".SCANNER[#Numero_SCR].Tipo;
       #Retval:=FILL(BVAL := #CERO, BLK => #Datos_fifo);
       SCATTER(IN := "Estado_inicializacion",
               OUT => #Inic_bits);


   END_REGION
   REGION comprobar_inicializacion
       // comprobamos si el scanner que estamos comprobando está en proceso de inicialización
       IF ((#Num_Inic >= 1) AND (#Num_Inic <= 8)) THEN
           // si tiene un numero de inicialización configurado, comprobamos si está activo
           IF (#Inic_bits[#Num_Inic] = true) THEN
               GOTO proceso_INIC;
           END_IF;
       END_IF;

   END_REGION

   REGION comprobar_etiqueta

       IF #EtiquetaTMP <= 0 THEN
           GOTO error_lectura;
       ELSE
           #Cola := #EtiquetaTMP MOD "ROUT_N_Colas";        // calculamos el numero de cola
       END_IF;
   END_REGION

   #Posicion_Etiqueta_TMP := "DB212_Cola_Activa".Cola[#Cola];

   // comprobamos si existe alguna etiqueta en esa cola

   elegir_db_busqueda:

       // si esa etiqueta no está dada de alta en las colas es que no está activa 
   IF #Posicion_Etiqueta_TMP = 0 THEN
       GOTO lectura_NENC;
   END_IF;


   REGION elegir_db_busqueda
       CASE #Posicion_Etiqueta_TMP OF
           1..1000:
               GOTO busca_1_999;
           1001..2000:
               GOTO busca_1k;
           2001..3000:
               GOTO busca_2k;
           3001..4000:
               GOTO busca_3k;
           ELSE

               GOTO lectura_NENC;
       END_CASE;
   END_REGION

   ////////////////////////////////////////////
   REGION busca_1_a_1000
   busca_1_999:
       IF #EtiquetaTMP = "DB201_RegEtiquetas_0001_1000".Reg_Etiqueta[#Posicion_Etiqueta_TMP].CDB THEN
           #Reg_Etiq_Temp := "DB201_RegEtiquetas_0001_1000".Reg_Etiqueta[#Posicion_Etiqueta_TMP];
           GOTO lectura_encontrada;
       ELSE
           #Posicion_Etiqueta_TMP := "DB201_RegEtiquetas_0001_1000".Reg_Etiqueta[#Posicion_Etiqueta_TMP].Posterior;
           GOTO elegir_db_busqueda;
       END_IF;
   END_REGION

   ////////////////////////////////////////////
   REGION busca_1001_a_2000
   busca_1k:
       #Posicion_Etiqueta_TMP := #Posicion_Etiqueta_TMP - 1000;
       IF #EtiquetaTMP = "DB202_RegEtiquetas_1001_2000".Reg_Etiqueta[#Posicion_Etiqueta_TMP].CDB THEN
           #Reg_Etiq_Temp := "DB202_RegEtiquetas_1001_2000".Reg_Etiqueta[#Posicion_Etiqueta_TMP];
           GOTO lectura_encontrada;
       ELSE
           #Posicion_Etiqueta_TMP := "DB202_RegEtiquetas_1001_2000".Reg_Etiqueta[#Posicion_Etiqueta_TMP].Posterior;
           GOTO elegir_db_busqueda;
       END_IF;
   END_REGION

   ////////////////////////////////////////////
   REGION busca_2001_a_3000
   busca_2k:
       #Posicion_Etiqueta_TMP := #Posicion_Etiqueta_TMP - 2000;
       IF #EtiquetaTMP = "DB203_RegEtiquetas_2001_3000".Reg_Etiqueta[#Posicion_Etiqueta_TMP].CDB THEN
           #Reg_Etiq_Temp := "DB203_RegEtiquetas_2001_3000".Reg_Etiqueta[#Posicion_Etiqueta_TMP];
           GOTO lectura_encontrada;
       ELSE
           #Posicion_Etiqueta_TMP := "DB203_RegEtiquetas_2001_3000".Reg_Etiqueta[#Posicion_Etiqueta_TMP].Posterior;
           GOTO elegir_db_busqueda;
       END_IF;

   END_REGION

   ////////////////////////////////////////////
   REGION busca_3001_a_4000
   busca_3k:
       #Posicion_Etiqueta_TMP := #Posicion_Etiqueta_TMP - 3000;
       IF #EtiquetaTMP = "DB204_RegEtiquetas_3001_4000".Reg_Etiqueta[#Posicion_Etiqueta_TMP].CDB THEN
           #Reg_Etiq_Temp := "DB204_RegEtiquetas_3001_4000".Reg_Etiqueta[#Posicion_Etiqueta_TMP];
           GOTO lectura_encontrada;
       ELSE
           #Posicion_Etiqueta_TMP := "DB204_RegEtiquetas_3001_4000".Reg_Etiqueta[#Posicion_Etiqueta_TMP].Posterior;
           GOTO elegir_db_busqueda;
       END_IF
       ;
   END_REGION

   REGION Especial_error_lectura
   error_lectura:
       #Reg_Etiq_Temp := "DB209_Reg_Etquetas_Esp_Activa".Reg_Etiqueta[1];
       #Datos_fifo.Orden := w#16#90;
       IF #Tipo_SCR = 2 THEN // tipo validación
           #Datos_fifo.Identificador := #Etiqueta;
           GOTO guardar_orden;
       END_IF;
       GOTO extraer_orden;
   END_REGION
   REGION Especial_NENC
   lectura_NENC:
       #Datos_fifo.Identificador := #Etiqueta;
       IF (#Tipo_SCR = 2) THEN
           #Datos_fifo.Orden := w#16#80;

           GOTO guardar_orden;
       END_IF;
       #Reg_Etiq_Temp := "DB209_Reg_Etquetas_Esp_Activa".Reg_Etiqueta[2];
       #Datos_fifo.Orden := w#16#A0;
       // hay dos casos posibles. si el escanner es normal extrae orden normal
       // si es de validacion de etiqueta, extrae el predeterminado
       GOTO extraer_orden;
   END_REGION
   REGION Especial_INIC
   proceso_INIC:
       #Reg_Etiq_Temp := "DB209_Reg_Etquetas_Esp_Activa".Reg_Etiqueta[3];
       #Datos_fifo.Orden := w#16#C0;
       GOTO extraer_orden;
   END_REGION
   REGION lectura_ok
   lectura_encontrada:
       #Datos_fifo.Identificador := #Etiqueta;
       IF #Tipo_SCR = 2 THEN
           #Datos_fifo.Orden := w#16#81;
           GOTO guardar_orden;
       ELSE
           #Datos_fifo.Orden := w#16#80;
           GOTO extraer_orden;
       END_IF;


   END_REGION

   REGION Extraer orden
   extraer_orden:
       #Datos_fifo.Identificador := #Etiqueta;
   // proceso extracción de la orden
   // miramos cual es el primer bit que tenemos que sacar de la orden
       #primer_bit := "DB912_Tipo_Scanner_Router".SCANNER[#Numero_SCR].Bit_Ini_Ordenes;
       #numero_bits := "DB912_Tipo_Scanner_Router".SCANNER[#Numero_SCR].N_Bits_Orden;
       #cont_aux := 0;
       #orden := #Datos_fifo.Orden;
       FOR #contador := #primer_bit TO (#primer_bit + #numero_bits - 1) DO
           #orden_aux[#cont_aux] := #Reg_Etiq_Temp.BIT_Orden[#contador];
           #cont_aux += 1;
       END_FOR;
       #Datos_fifo.Orden := #orden;
       ;
   END_REGION

   REGION Guardar_Orden
   guardar_orden:
       // miramos si ya hay algo en la fifo
       "FC571_Leer_Datos_Fifo"(DB_FIFO_Ordenes:="ROUT_NDB_FIFO_Odr_SCR",
                               Num_Scanner:=#Numero_SCR,
                               Long_FIFO:=1,
                               Posicion_FIFO:=1,
                               Datos_Scanner_Cruce=>#datos_actuales_fifo);

       IF #datos_actuales_fifo.Orden <> 0 THEN
           #Datos_fifo.Orden := w#16#FF;
       END_IF;
       "FC572_Guardar_Datos_Fifo"(DB_FIFO_Ordenes:="ROUT_NDB_FIFO_Odr_SCR",
                                  Num_Scanner:=#Numero_SCR,
                                  Long_FIFO:=1,
                                  Posicion_FIFO:=1,
                                  Datos_Scanner_Cruce:=#Datos_fifo);

       // lo ultimo es borrar la N de la nueva lectura en el db211   ;
       // 
       "DB211_Lecturas_Scanner".Lec_Scanner[#Numero_SCR].Lectura_SCR[0]:= l#0;



   END_REGION
END_FUNCTION

FUNCTION "FC781_Evento_ORDE" : Void   // FC781, LAD
{ S7_Optimized_Access := 'TRUE' }
// stored: AutoNumber false, SetENOAutomatically false
   VAR_INPUT
      mensaje : Int;
   END_VAR
   VAR_TEMP
      pos_mesa : Int;
      numero_mesa : Int;
      pos_sali : Int;
      valor_sali : Int;
   END_VAR
BEGIN

REGION Network 1 (SCL)
   // EXTRAEMOS EL VALOR DEL NUMERO DE MESA
   // 
   #pos_mesa := FIND(IN1 := "DB199_eventos_convertidos".evento[#mensaje], IN2 := '[MESA]');

   STRG_VAL(IN := "DB199_eventos_convertidos".evento[#mensaje],
            FORMAT := 0,
            P := (#pos_mesa + 6), // +6 por lo que ocupa el atributo ['SSCC]'
            OUT => #numero_mesa);

   // EXTRAEMOS EL VALOR DEL ATRIBUTO SALI
   #pos_sali := FIND(IN1 := "DB199_eventos_convertidos".evento[#mensaje], IN2 := '[SALI]');

   STRG_VAL(IN := "DB199_eventos_convertidos".evento[#mensaje],
            FORMAT := 0,
            P := (#pos_sali + 6), // +6 por lo que ocupa el atributo ['SSCC]'
            OUT => #valor_sali);

   //ASIGNAMOS EL VALOR EL EL DB
   // 
   "DB841_Recepcion".Mesa[#numero_mesa-CTE_OffsetMesa].Auxiliar_04 := #valor_sali + 3000;
END_REGION
END_FUNCTION

FUNCTION "FC782_Evento_RUES" : Void   // FC782, LAD
{ S7_Optimized_Access := 'FALSE' }
// stored: AutoNumber false, SetENOAutomatically false
   VAR_INPUT
      mensaje : Int;   // indice del array que estamos extrayendo
   END_VAR
   VAR_TEMP
      Existe_ruta : Bool;
      retval : Int;
      pos_SSCC : UInt;
      cero : Byte;
      destinos : Array[0..9] of UInt;
      registro_etiqueta : "ROUT_Reg_Etiqueta";
      orden_desvio : Byte;
      desvio_bits AT orden_desvio : Array[1..8] of Bool;
      posicion : Int;
      pos_ruta : Int;
      posicion_mesa : Int;
      posicion_db : Int;
      desvio : Int;
      scanner : UInt;
      bit_ini : Int;
      n_bits : Int;
      contador_aux : Int;
      contador : Int;
      posicion_BBDD : UInt;
      Atributo_rues : String[4];
   END_VAR
BEGIN

REGION Network 1 (SCL): INICIALIZACIONES
   REGION inicializacion

       // inicializamos las variables
       // 

       #retval := FILL(BVAL := #cero, BLK => #registro_etiqueta); // el registro de la etiqueta temporal
       #retval := FILL(BVAL := #cero, BLK => #destinos); // los datos temporales de los destinos
       #orden_desvio := 0;
       #Existe_ruta := false;

   END_REGION
END_REGION

REGION Network 2 (SCL): EXTRAEMOS DEL MENSAJE LOS DESTINOS

   // miramos si en el mensaje nos han llegado destinos que extraer
   #posicion := FIND(IN1 := "DB199_eventos_convertidos".evento[#mensaje], IN2 := '[DEST]');
   IF #posicion <> 0 THEN    // iniciamos la estracción de las mesas que pertenecen a la ruta
           // si solamente se ejecuta el proceso una vez en el mensaje no es necesario realizar esta operación de sustituir el atributo DEST
       "DB199_eventos_convertidos".evento[#mensaje] := REPLACE(IN1 := "DB199_eventos_convertidos".evento[#mensaje], IN2 := '[dest]', L := 6, P := #posicion);
       #pos_ruta := 0;
       #Existe_ruta := 1;
       // temporalmente ponemos las rutas a cero
       WHILE #Existe_ruta DO
           #posicion := FIND(IN1 := "DB199_eventos_convertidos".evento[#mensaje], IN2 := '[MESA]');
           IF #posicion <> 0 THEN
               STRG_VAL(IN := "DB199_eventos_convertidos".evento[#mensaje],
                        FORMAT := 0,
                        P := (#posicion + 6),
                        OUT => #destinos[#pos_ruta]);
               #pos_ruta += 1; // incrementamos la posición en el array para seguir guardando
               // las mesas ya extraidas, las ponemos en minucula para seguir buscando las siguientes mesas sin eliminar parcialmente el mensaje
               "DB199_eventos_convertidos".evento[#mensaje] := REPLACE(IN1 := "DB199_eventos_convertidos".evento[#mensaje], IN2 := '[mesa]', L := 6, P := #posicion);
           ELSE
               #Existe_ruta := 0;
               EXIT;
           END_IF;
       END_WHILE;
   END_IF;
   // aqui tenemos que incluir la conversión de las mesas el los bits de cruce
END_REGION

REGION Network 3 (SCL): generación de los bits de cruce
   REGION generar_bits_cruce
       #posicion_mesa := 0;
       #posicion_db := 0;

       WHILE #destinos[#posicion_mesa] <> 0 DO
           // Statement section WHILE

           WHILE (("DB913_Router_DestinoDesvio".DestinoDesvios[#posicion_db].Destino <> 0) AND (#posicion_db <= "ROUT_Max_Destinos")) DO
               IF (#destinos[#posicion_mesa] = "DB913_Router_DestinoDesvio".DestinoDesvios[#posicion_db].Destino) THEN
                   // si coincide la mesa con uno de los destinos
                   #desvio := 0;
                   WHILE (("DB913_Router_DestinoDesvio".DestinoDesvios[#posicion_db].Desvios[#desvio].SCR <> 0) AND (#desvio <= "ROUT_Max_Destinos")) DO
                       #scanner := "DB913_Router_DestinoDesvio".DestinoDesvios[#posicion_db].Desvios[#desvio].SCR;
                       #orden_desvio := "DB913_Router_DestinoDesvio".DestinoDesvios[#posicion_db].Desvios[#desvio].Bits;
                       #bit_ini := "DB912_Tipo_Scanner_Router".SCANNER[#scanner].Bit_Ini_Ordenes;
                       #n_bits := "DB912_Tipo_Scanner_Router".SCANNER[#scanner].N_Bits_Orden;

                       // aqui mediante un for vamos escribiendo los bits donde corresponden
                       #contador_aux := 1;
                       FOR #contador := #bit_ini TO (#bit_ini + #n_bits - 1) DO
                           #registro_etiqueta.BIT_Orden[#contador] := #desvio_bits[#contador_aux];
                           #contador_aux += 1;

                       END_FOR;
                       #desvio += 1; // nos desplazamos el siguiente desvio
                   END_WHILE;

               END_IF;
               #posicion_db += 1; //nos desplazamos hasta el siguiente destino
           END_WHILE;
           #posicion_mesa += 1; // nos desplazamos a la siguiente mesa destino de la ruta
           #posicion_db := 0; // inicializamos a cero la busqueda dentro del DB de destinos

       END_WHILE;

   END_REGION
END_REGION

REGION Network 4 (SCL): volcado al DB de datos
   #pos_SSCC := FIND(IN1 := "DB199_eventos_convertidos".evento[#mensaje], IN2 := '[ETES]');
   // extraemos el dato de qué etiqueta especial se trata
   // 

   #Atributo_rues:=MID(IN := "DB199_eventos_convertidos".evento[#mensaje], L := 4, P := (#pos_SSCC + 6));

   // elección de la posición de volcado
   // 
   IF (#Atributo_rues = 'ERRR') THEN
       // especiales registro 1
       "DB209_Reg_Etquetas_Esp_Activa".Reg_Etiqueta[1] := #registro_etiqueta;
   ELSE
       IF (#Atributo_rues = 'NENC') THEN
           // especiales registro 2
           "DB209_Reg_Etquetas_Esp_Activa".Reg_Etiqueta[2] := #registro_etiqueta;
       ELSE
           IF (#Atributo_rues = 'INIC') THEN
               // especiales registro 3
               "DB209_Reg_Etquetas_Esp_Activa".Reg_Etiqueta[3] := #registro_etiqueta;
           END_IF;
       END_IF;
   END_IF;
END_REGION
END_FUNCTION

FUNCTION "FC783_Evento_BOET" : Void   // FC783, LAD
{ S7_Optimized_Access := 'FALSE' }
// stored: AutoNumber false, SetENOAutomatically false
   VAR_INPUT
      mensaje : Int;   // indice del array que estamos extrayendo
   END_VAR
   VAR_TEMP
      cero : Byte;
      retval : Int;
      pos_SSCC : UInt;
      Etiqueta_a_eliminar : ULInt;
      posicion_a_eliminar : UInt;
      cola : UInt;
      dato_actual_cola : UInt;
      pos_DB : UInt;
      registro_anterior : UInt;
      registro_siguiente : UInt;
      registro_etiqueta_limpio : "ROUT_Reg_Etiqueta";
   END_VAR
BEGIN

REGION Network 1 (SCL): INICIALIZACIONES
   REGION inicializacion

       // inicializamos las variables
       // 

       #retval := FILL(BVAL := #cero, BLK => #registro_etiqueta_limpio); // el registro de la etiqueta temporal



   END_REGION
END_REGION

REGION Network 2 (SCL): RECOJO Y CONVIERTO EL VALOR DE LA EITQUETA
   // buscamos donde empieza el SSCC en el mensaje y lo convertimos
   // 
   #pos_SSCC := FIND(IN1 := "DB199_eventos_convertidos".evento[#mensaje], IN2 := '[SSCC]');

   STRG_VAL(IN := "DB199_eventos_convertidos".evento[#mensaje],
            FORMAT := 0,
            P := (#pos_SSCC + 6), // +6 por lo que ocupa el atributo ['SSCC]'
            OUT => #Etiqueta_a_eliminar
   );

   // buscamos la etiqueta en la BBDD

   "FC715_Router_BuscarEtiqueta_Lint"(Etiqueta :=#Etiqueta_a_eliminar ,
                                      Posicion_BBDD => #posicion_a_eliminar);


   // si la posición a eliminar es 0, es que no existe ya en la BBDD y salimos de la función
   // 
   IF #posicion_a_eliminar = 0 THEN
       RETURN;
   END_IF;

     // si la hemos encontrado, además de eliminar la etiqueta, tenemos que mantener la coherencia
     // en el sistema de colas
     // para eso tenemos que mirar la posicón anterior y siguiente
     // 
     //
     //CALCULAMOS LA COLA A LA QUE PERTENECE LA ETIQUETA 
   #cola :=#Etiqueta_a_eliminar MOD "ROUT_N_Colas";


   REGION elegir_db_busqueda
       CASE #posicion_a_eliminar OF
           1..1000:
               #pos_DB := #posicion_a_eliminar;
               #registro_anterior:="DB201_RegEtiquetas_0001_1000".Reg_Etiqueta[#pos_DB].Anterior;
               #registro_siguiente:="DB201_RegEtiquetas_0001_1000".Reg_Etiqueta[#pos_DB].Posterior;
               // ahora que ya he sacado los datos necesarios limpio el registro
               "DB201_RegEtiquetas_0001_1000".Reg_Etiqueta[#pos_DB] := #registro_etiqueta_limpio;
               IF ((#registro_anterior = 0) AND (#registro_siguiente = 0)) THEN
                   "DB212_Cola_Activa".Cola[#cola] := 0;
                   RETURN;
               END_IF;

           1001..2000:
               #pos_DB := #posicion_a_eliminar - 1000;
               #registro_anterior := "DB202_RegEtiquetas_1001_2000".Reg_Etiqueta[#pos_DB].Anterior;
               #registro_siguiente := "DB202_RegEtiquetas_1001_2000".Reg_Etiqueta[#pos_DB].Posterior;
               "DB202_RegEtiquetas_1001_2000".Reg_Etiqueta[#pos_DB] := #registro_etiqueta_limpio;
               IF ((#registro_anterior = 0) AND (#registro_siguiente = 0)) THEN
                   "DB212_Cola_Activa".Cola[#cola] := 0;
                   RETURN;
               END_IF;

           2001..3000:
               #pos_DB := #posicion_a_eliminar - 2000;
              #registro_anterior:= "DB203_RegEtiquetas_2001_3000".Reg_Etiqueta[#pos_DB].Anterior ;
              #registro_siguiente:= "DB203_RegEtiquetas_2001_3000".Reg_Etiqueta[#pos_DB].Anterior;
               "DB203_RegEtiquetas_2001_3000".Reg_Etiqueta[#pos_DB] := #registro_etiqueta_limpio;
               // si los dos campos son 0 es que soy la unica etiqueta de la cola
               IF ((#registro_anterior = 0) AND (#registro_siguiente = 0)) THEN
                   "DB212_Cola_Activa".Cola[#cola] := 0;
                   RETURN;
               END_IF;
           3001..4000:
               #pos_DB := #posicion_a_eliminar - 3000;
               #registro_anterior := "DB204_RegEtiquetas_3001_4000".Reg_Etiqueta[#pos_DB].Anterior;
               #registro_siguiente := "DB204_RegEtiquetas_3001_4000".Reg_Etiqueta[#pos_DB].Posterior;
               "DB204_RegEtiquetas_3001_4000".Reg_Etiqueta[#pos_DB] := #registro_etiqueta_limpio;
               // si los dos campos son 0 es que soy la unica etiqueta de la cola
               IF ((#registro_anterior = 0) AND (#registro_siguiente = 0)) THEN
                   "DB212_Cola_Activa".Cola[#cola] := 0;
                   RETURN;
               END_IF;

               RETURN;
       END_CASE;
   END_REGION

   // si alguno de los dos datos es distinto de cero, tengo que recomponer la cola modificando
   // los registos de las etiquetas anteriores, posteriores y si procede la cola.
   // 

   IF #registro_anterior = 0 THEN
       // soy la primera de la cola y tengo que hacer que la que va despues de mi sea la primera de la cola

       "DB212_Cola_Activa".Cola[#cola] := #registro_siguiente;
   END_IF;

   //recomponemos registro anterior en la siguiente etiqueta
       REGION elegir_db_busqueda
           CASE #registro_siguiente OF
               0:
                   ;
               1..1000:
                   #pos_DB := #registro_siguiente;
                   "DB201_RegEtiquetas_0001_1000".Reg_Etiqueta[#pos_DB].Anterior := #registro_anterior;


               1001..2000:
                   #pos_DB := #registro_siguiente - 1000;
                   "DB202_RegEtiquetas_1001_2000".Reg_Etiqueta[#pos_DB].Anterior := #registro_anterior;

               2001..3000:
                   #pos_DB := #registro_siguiente - 2000;
                   "DB203_RegEtiquetas_2001_3000".Reg_Etiqueta[#pos_DB].Anterior := #registro_anterior;


               3001..4000:
                   #pos_DB := #registro_siguiente - 3000;
                   "DB204_RegEtiquetas_3001_4000".Reg_Etiqueta[#pos_DB].Anterior := #registro_anterior;


           END_CASE;
       END_REGION
       //recomponemos registro siguiente en la siguiente anterior
       REGION elegir_db_busqueda
           CASE #registro_anterior OF
               0:
                   ;
               1..1000:
                   #pos_DB := #registro_anterior;
                   "DB201_RegEtiquetas_0001_1000".Reg_Etiqueta[#pos_DB].Posterior := #registro_siguiente;
                   RETURN;

               1001..2000:
                   #pos_DB := #registro_anterior - 1000;
                   "DB202_RegEtiquetas_1001_2000".Reg_Etiqueta[#pos_DB].Posterior := #registro_siguiente;
                   RETURN;
               2001..3000:
                   #pos_DB := #registro_anterior - 2000;
                   "DB203_RegEtiquetas_2001_3000".Reg_Etiqueta[#pos_DB].Posterior := #registro_siguiente;
                   RETURN;

               3001..4000:
                   #pos_DB := #registro_anterior - 3000;
                   "DB204_RegEtiquetas_3001_4000".Reg_Etiqueta[#pos_DB].Posterior := #registro_siguiente;
                   RETURN;


           END_CASE;
       END_REGION
END_REGION
END_FUNCTION

FUNCTION "FC784_Evento_INIR" : Void   // FC784, LAD
{ S7_Optimized_Access := 'FALSE' }
// stored: AutoNumber false, SetENOAutomatically false
   VAR_INPUT
      mensaje : Int;
   END_VAR
   VAR_TEMP
      numero : Int;
      numero_inicializacion : Int;
      pos_habi : Int;
      habi : String[2];
      ESTADO_HABI : Byte;
      ESTADO_HABI_BITS AT ESTADO_HABI : Array[1..8] of Bool;
      MENSAJE_EMI : String[50];
      Numero_string : String[1];
      atributo_habi : String[2];
      i : Int;
      longitud : Int;
   END_VAR
BEGIN

REGION Network 1 (SCL)
   // EXTRAEMOS EL VALOR DEL NUMERO DE LA INICIALIZACIÓN QUE TENEMOS QUE HABILITAR
   // 
   #numero := FIND(IN1 := "DB199_eventos_convertidos".evento[#mensaje], IN2 := '[NUME]');

   STRG_VAL(IN := "DB199_eventos_convertidos".evento[#mensaje],
            FORMAT := 0,
            P := (#numero + 6), // +6 por lo que ocupa el atributo ['SSCC]'
            OUT => #numero_inicializacion);

   // COMPROBAMOS LA VALIDED DEL NUMERO DE INICIALIZACIÓN. ACTUALMENTE EL MÁXIMO ES 8
   // 

   IF #numero_inicializacion > 8 THEN
       // formatear el mensaje de inicialización no posible
       // 

       #Numero_string := DELETE(IN := (INT_TO_STRING(IN := #numero_inicializacion)), L := 1, P := 1);
       // 
       #MENSAJE_EMI := CONCAT(IN1 := '{INI![NUME]', IN2 := #Numero_string, IN3 := '[HABI]NO[MOTI]NOOK', IN4 := "DB921_DATOS_FECHA_HORA".TIME_STAMP, IN5 := '}');

       REGION emision_mensaje
           // miramos donde tenemos que emitir el mensaje
           IF "ROUT_X_CONEX_JDT1" = FALSE THEN
               REGION buscar en JDT2                
                   FOR #i := 0 TO 100 BY 1 DO
                       #longitud := LEN("DB197_eventos_generados_routing_JDT2".evento[#i]);
                       IF #longitud = 0 THEN
                           "DB197_eventos_generados_routing_JDT2".evento[#i] := #MENSAJE_EMI;
                           RETURN;
                       END_IF;
                   END_FOR;
                   // si ha acabado el for sin encontrar sitio no puedo emititir y salgo de la funcion
                   RETURN;
               END_REGION
               ;
           ELSE
               REGION buscar en JDT1
                   FOR #i := 0 TO 100 BY 1 DO
                       #longitud := LEN("DB198_eventos_generados_routing_JDT1".evento[#i]);
                       IF #longitud = 0 THEN
                           "DB198_eventos_generados_routing_JDT1".evento[#i] := #MENSAJE_EMI;
                           RETURN;
                       END_IF;
                   END_FOR;
                   // si ha acabado el for sin encontrar sitio no puedo emititir y salgo de la funcion
                   RETURN;

               END_REGION
           END_IF;
       END_REGION
       ;
   END_IF;

   // EXTRAEMOS EL VALOR DEL ATRIBUTO HABI
   #pos_habi := FIND(IN1 := "DB199_eventos_convertidos".evento[#mensaje], IN2 := '[HABI]');

   #habi:=MID(IN:="DB199_eventos_convertidos".evento[#mensaje], L:=2, P:=#pos_habi+6);


   IF #habi = 'SI' THEN  //TENEMOS QUE HABILITAR LA INICIALIZACIÓN

       #ESTADO_HABI := "Estado_inicializacion";     // PRIMERO COGEMOS EL VALOR QUE TIENEN LAS MEMORIAS ACTUALENTE
       #ESTADO_HABI_BITS[#numero_inicializacion] := TRUE;
       "Estado_inicializacion" := #ESTADO_HABI;    //VOLVEMOS A VOLCAR EL ESTADO EN LA PALABRA GLOBAL

       // FORMATEAMOS EL MENSAJE



       #Numero_string := DELETE(IN := (INT_TO_STRING(IN := #numero_inicializacion)), L := 1, P := 1);

       #MENSAJE_EMI := CONCAT(IN1 := '{INI![NUME]', IN2 := #Numero_string, IN3 := '[HABI]SI', IN4 := "DB921_DATOS_FECHA_HORA".TIME_STAMP,IN5 := '}');

   ELSIF #habi = 'NO' THEN

       #ESTADO_HABI := "Estado_inicializacion"; // PRIMERO COGEMOS EL VALOR QUE TIENEN LAS MEMORIAS ACTUALENTE
       #ESTADO_HABI_BITS[#numero_inicializacion] := FALSE;
       "Estado_inicializacion" := #ESTADO_HABI;   //VOLVEMOS A VOLCAR EL ESTADO EN LA PALABRA GLOBAL

       // FORMATEAMOS EL MENSAJE



       #Numero_string := DELETE(IN := (INT_TO_STRING(IN := #numero_inicializacion)), L := 1, P := 1);

       #MENSAJE_EMI := CONCAT(IN1 := '{INI![NUME]', IN2 := #Numero_string, IN3 := '[HABI]NO', IN4 := "DB921_DATOS_FECHA_HORA".TIME_STAMP, IN5 := '}');

   ELSIF #habi = '??' THEN
       // MIRAMOS SI ESTÁ HABILITADO O NO PARA FORMATEAR EL MENSAJE
       #ESTADO_HABI := "Estado_inicializacion"; // PRIMERO COGEMOS EL VALOR QUE TIENEN LAS MEMORIAS ACTUALENTE

       IF #ESTADO_HABI_BITS[#numero_inicializacion] = TRUE THEN
           #atributo_habi := 'SI';
       ELSE
           #atributo_habi := 'NO';
       END_IF;


       // FORMATEAMOS EL MENSAJE


       #Numero_string := DELETE(IN := (INT_TO_STRING(IN := #numero_inicializacion)), L := 1, P := 1);

       #MENSAJE_EMI := CONCAT(IN1 := '{INI![NUME]', IN2 := #Numero_string, IN3 := '[HABI]',IN4:=#atributo_habi, IN5 := "DB921_DATOS_FECHA_HORA".TIME_STAMP, IN6 := '}');
       ;
   END_IF;


   REGION emision_mensaje
       // miramos donde tenemos que emitir el mensaje
       IF "ROUT_X_CONEX_JDT1" = FALSE THEN
           REGION buscar en JDT2                
               FOR #i := 0 TO 100 BY 1 DO
                       #longitud := LEN("DB197_eventos_generados_routing_JDT2".evento[#i]);
                       IF #longitud = 0 THEN
                           "DB197_eventos_generados_routing_JDT2".evento[#i]:=#MENSAJE_EMI;
                           RETURN;
                       END_IF;
                   END_FOR;
                   // si ha acabado el for sin encontrar sitio no puedo emititir y salgo de la funcion
                   RETURN;
               END_REGION
               ;
           ELSE
               REGION buscar en JDT1
                   FOR #i := 0 TO 100 BY 1 DO
                       #longitud := LEN("DB198_eventos_generados_routing_JDT1".evento[#i]);
                       IF #longitud = 0 THEN
                           "DB198_eventos_generados_routing_JDT1".evento[#i] := #MENSAJE_EMI;
                           RETURN;
                       END_IF;
                   END_FOR;
                   // si ha acabado el for sin encontrar sitio no puedo emititir y salgo de la funcion
                       RETURN;

               END_REGION
           END_IF;
   END_REGION
END_REGION
END_FUNCTION

FUNCTION "FC818_Mensaje_BBDD_Routing_Llena" : Void   // FC818, LAD
{ S7_Optimized_Access := 'FALSE' }
// stored: AutoNumber false, SetENOAutomatically false
   VAR_INPUT
      Etiqueta : ULInt;
      Envio_JDT2 : Bool;
   END_VAR
   VAR_TEMP
      Guardar_AR1 : DWord;
      DBEventos : Word;   // Numero del DB de Eventos
      PunteroEventos : DWord;   // Puntero al DB de Eventos
      MaxBytes : UInt;
      NDB_Eventos_Emi : UInt;
      NumBytes : UInt;   // Numero de Bytes existentes en el DB de Eventos
      etiqueta_string : String;
      indice : Int;
      longitud : Int;
      posicion : Int;
      i : Int;
      codigo_string : String[20];
   END_VAR
BEGIN

REGION Network 1 (SCL)
   // buscamos hueco en el db donde vamos a escribir los eventos antes de empezar la conversión
   // 


   IF #Envio_JDT2    = true THEN
       REGION buscar en JDT2

           #posicion := -1;
           FOR #i := 0 TO 100 BY 1 DO
               #longitud := LEN("DB197_eventos_generados_routing_JDT2".evento[#i]);
               IF #longitud = 0 THEN
                   #posicion := #i;
                   EXIT;
               END_IF;
           END_FOR;

           // si no hay sitio para escribir salimos del bloque
           IF #posicion = -1 THEN
               RETURN;
           END_IF;
       END_REGION
       ;
   ELSE
       REGION buscar en JDT1

           #posicion := -1;
           FOR #i := 0 TO 100 BY 1 DO
               #longitud := LEN("DB198_eventos_generados_routing_JDT1".evento[#i]);
               IF #longitud = 0 THEN
                   #posicion := #i;
                   EXIT;
               END_IF;
           END_FOR;

           // si no hay sitio para escribir salimos del bloque
           IF #posicion = -1 THEN
               RETURN;
           END_IF;
       END_REGION
   END_IF;
END_REGION

REGION Network 2 (SCL): formatear el evento


   #codigo_string := DELETE(IN := (ULINT_TO_STRING(IN := #Etiqueta)), L := 1, P := 1);
   // concatenamos el mensaje 
   // 
   IF #Envio_JDT2= true THEN

       "DB197_eventos_generados_routing_JDT2".evento[#posicion] := CONCAT(IN1 := '{WARN[RUET]', IN2 := #codigo_string, IN3 := '[ERRO]BBDD[MOTI]FULL',  IN4 := "DB921_DATOS_FECHA_HORA".TIME_STAMP, IN5 := '}');

